		// 3. Lateral nicht OK: Querrichtung bevorzugen, Einfahrt gedrosselt
		ELSIF (PosLatOK = FALSE) THEN
			IF ePocketOrientation = ePocketX THEN
				FB_Positionsregler(targetPos := targetPos, actualPos := actualPos,
								KPX := 0.2 * KPX, KPY := KPY, KIX := 0.2 * KIX, KIY := KIY,
								vXCartesianToMotors     => targetSpeed_Robot.reX,
								vYCartesianToMotors     => targetSpeed_Robot.reY,
								vThetaCartesianToMotors => targetSpeed_Robot.reWinkel);
			ELSE
				FB_Positionsregler(targetPos := targetPos, actualPos := actualPos,
								KPX := KPX, KPY := 0.1 * KPY, KIX := KIX, KIY := 0.1 * KIY,
								vXCartesianToMotors     => targetSpeed_Robot.reX,
								vYCartesianToMotors     => targetSpeed_Robot.reY,
								vThetaCartesianToMotors => targetSpeed_Robot.reWinkel);
			END_IF
			GVL_Datatransfer23.inStatus := RobotStatus.laufend;
		
		// 4. Normalbetrieb
		ELSIF (Gripper.slider = TRUE) THEN
			
			IF ePocketOrientation = ePocketX THEN
				FB_Positionsregler(targetPos := targetPos, actualPos := actualPos,
								KPX := KPX, KPY := KPY, KIX := KIX, KIY := KIY,
								vXCartesianToMotors     => targetSpeed_Robot.reX,
								vYCartesianToMotors     => targetSpeed_Robot.reY,
								vThetaCartesianToMotors => targetSpeed_Robot.reWinkel);
			ELSE
				FB_Positionsregler(targetPos := targetPos, actualPos := actualPos,
								KPX := KPX, KPY := KPY, KIX := KIX, KIY := 2*KIY,
								vXCartesianToMotors     => targetSpeed_Robot.reX,
								vYCartesianToMotors     => targetSpeed_Robot.reY,
								vThetaCartesianToMotors => targetSpeed_Robot.reWinkel);
			END_IF			
			GVL_Datatransfer23.inStatus := RobotStatus.laufend;
		
		// 5. Ziel erreicht
		ELSE
			FB_Positionsregler(targetPos := targetPos, actualPos := actualPos,
								vXCartesianToMotors     => targetSpeed_Robot.reX,
								vYCartesianToMotors     => targetSpeed_Robot.reY,
								vThetaCartesianToMotors => targetSpeed_Robot.reWinkel);
								targetSpeed_Robot.reY := 0;
								targetSpeed_Robot.reX := 0;
								targetSpeed_Robot.reWinkel := 0;
			GVL_Datatransfer23.inStatus := RobotStatus.zielErreicht;
		END_IF
	
	END_CASE
	
//enableMotorControl := FALSE;
/////////////////////////////////////////////////////////////////////////////////////////////////////////
// Drehzahlregler
/////////////////////////////////////////////////////////////////////////////////////////////////////////
FB_Drehzahlregler(targetVelX			:= targetSpeed_Robot.reX,
					targetVelY 			:= targetSpeed_Robot.reY, 
					tragetVelTheta		:= targetSpeed_Robot.reWinkel,
					enable 				:= enableMotorControl,
					bumper 				:= bumper,
					MotorReset 			:= FALSE,
					actualVelMotor1 	:= -velWheel1, 
					actualVelMotor2 	:= -velWheel2, 
					actualVelMotor3 	:= -velWheel3,
					enableToMotor1 		=> enableToMotor1,
					enableToMotor2 		=> enableToMotor2,
					enableToMotor3 		=> enableToMotor3,
					velocityToMotor1	=> velocityToMotor1, 
					velocityToMotor2	=> velocityToMotor2,
					velocityToMotor3	=> velocityToMotor3);

ACTION ACT_Drehzahlerfassung:
//Einlesen der Istwerte
//Motorstrom von der Klemme auslesen und umrechnen
Motor1current := UINT_TO_INT(currentfromMotor1);	//Umwandlung des Unsinged Integers in ein Integerwert
Motor2current := UINT_TO_INT(currentfromMotor2);
Motor3current := UINT_TO_INT(currentfromMotor3);

//Berechnung der Radgeschwindigkeit mit berücksichtigung des Getriebes
velWheel1 := -(UINT_TO_INT(n1fromMotor) / maxKlemmeDrehzahlMessung*maxMotorRPM/60*ue*2*PI*rWheel);
velWheel2 := -(UINT_TO_INT(n2fromMotor) / maxKlemmeDrehzahlMessung*maxMotorRPM/60*ue*2*PI*rWheel);
velWheel3 := -(UINT_TO_INT(n3fromMotor) / maxKlemmeDrehzahlMessung*maxMotorRPM/60*ue*2*PI*rWheel);
END_ACTION

METHOD ATAN2 : LREAL
VAR_INPUT
    y : LREAL;
    x : LREAL;
END_VAR

VAR
    raw_angle : LREAL;
END_VAR

IF x = 0.0 THEN
    IF y > 0.0 THEN
        ATAN2 := 90.0;
    ELSIF y < 0.0 THEN
        ATAN2 := 270.0;
    ELSE
        ATAN2 := 0.0;
    END_IF;

ELSE
    raw_angle := ATAN(y / x) * (180.0 / PI);

    IF x > 0.0 THEN
        ATAN2 := raw_angle;
    ELSE
        ATAN2 := raw_angle + 180.0;
    END_IF;

    IF ATAN2 < 0.0 THEN
        ATAN2 := ATAN2 + 360.0;
    END_IF;
END_IF;
END_METHOD

METHOD Beobachter
VAR_INPUT
	wheelSpeed : WheelVelocity;
	cameraData : CameraConnectionUDP;
	RobotIndex : INT;
END_VAR
VAR_OUTPUT
	eastPos : sPosition := (reX := 0, reY := 0, reWinkel := 0);
END_VAR
VAR CONSTANT
	// === BEOBACHTER-PARAMETER => Großer Gain bedeutet hohes vertrauen in Kamera ===
	L_Gain					: REAL := 1.0;			// Luenberger Gain für X 		(0.0001-0.1)

	CYCLETIME 				: LREAL := 0.00033333;  // Cycletime des Motortasks
	CAMERA_DELAY			: REAL 	:= 0.1;
	BUFFWE_LENGTH			: INT 	:= 500;
	CAMERA_ERROR_THRESHOLD	: REAL 	:= 5.0;		// Fehlergrenze
	CAMERA_TIMEOUT			: LREAL := 30.0;		// Timeout in Sekunden
END_VAR

VAR_STAT
	bufferWheelSpeed	: ARRAY[0..BUFFWE_LENGTH] OF WheelVelocity;			// Speichern der letzten 300 Motorwerte (entspricht 100 ms -> Delay)
	prefCamPos			: sPosition;			// vorherige Kamera Position
	camPos				: sPosition;
	modelPos			: sPosition;
	CurrentTime			: LREAL;
	CameraTimestamp		: LREAL;
	actualError			: LREAL;				// Kamerafehler
	bufferIdx			: INT := 0;
	init				: BOOL;
END_VAR
VAR
	P_currentState 		: ARRAY[1..9] OF LREAL;	// Wär später für Kalmann	
	i					: INT;					// Iterrationsvariable
	averageWheelSpeed 	: WheelVelocity;
	x_estimated			: INT;
	angleError			: LREAL;
	idx					: INT;
	steps				: INT;
	startIdx			: INT;
	variableGain		: LREAL;
END_VAR
// Am anfang einmal die Kammeraposition direkt übertragen
IF init = TRUE THEN
	// Wenn ein guter Kamerawert gefunden wurde direkt einmal übertragen
	IF cameraData.robotPosition[RobotIndex].e < CAMERA_ERROR_THRESHOLD THEN
		camPos.reX 			:= cameraData.robotPosition[RobotIndex].x;
		camPos.reY 			:= cameraData.robotPosition[RobotIndex].y;
		camPos.reWinkel 	:= cameraData.robotPosition[RobotIndex].theta;
		actualError			:= cameraData.robotPosition[RobotIndex].e;
		prefCamPos 	:= camPos;
		modelPos	:= camPos;
		eastPos		:= camPos;
		
		init := FALSE;
	END_IF
ELSE
	/////////////////////////////////////////////////////////////////////////////////////////////////////////
	// Radwerte in FIFO abspeichern
	/////////////////////////////////////////////////////////////////////////////////////////////////////////
	bufferWheelSpeed[bufferIdx] := wheelSpeed;
	bufferIdx := (bufferIdx + 1) MOD BUFFWE_LENGTH;
	
	/////////////////////////////////////////////////////////////////////////////////////////////////////////
	// Modell Propagieren
	/////////////////////////////////////////////////////////////////////////////////////////////////////////
	propagate_state(
				X_Start 	:= modelPos,
				wheelSpeed 	:= wheelSpeed, 
				P_Start 	:= P_currentState,
				deltaT 		:= CYCLETIME,
				X_Predict 	=> modelPos,
				P_Predict 	=> P_currentState
			);
	CurrentTime := CurrentTime + CYCLETIME;	// Zeit weiter laufen lassen, wenn keine Kameradaten kommen
	
	/////////////////////////////////////////////////////////////////////////////////////////////////////////
	// Kameradaten verarbeiten
	/////////////////////////////////////////////////////////////////////////////////////////////////////////
	
	// Kammeraposition erst validieren
	IF cameraData.robotPosition[RobotIndex].e > CAMERA_ERROR_THRESHOLD OR
		// Prüfen ob neue Kameraposition
	   ((prefCamPos.reX 	 = cameraData.robotPosition[RobotIndex].x)	AND
		(prefCamPos.reY 	 = cameraData.robotPosition[RobotIndex].y) 	AND
		(prefCamPos.reWinkel = cameraData.robotPosition[RobotIndex].theta)) THEN
			
			// Falls keine neue Kameraposition erscheint, auch die Kamera vorwärtspropagieren
			propagate_state(
					X_Start 	:= camPos,
					wheelSpeed 	:= wheelSpeed, 
					P_Start 	:= P_currentState,
					deltaT 		:= CYCLETIME,
					X_Predict 	=> camPos,
					P_Predict 	=> P_currentState
				);
	ELSE
		// Falls Kameraposition gut nehmen
		camPos.reX 			:= cameraData.robotPosition[RobotIndex].x;
		camPos.reY 			:= cameraData.robotPosition[RobotIndex].y;
		camPos.reWinkel 	:= cameraData.robotPosition[RobotIndex].theta;
		actualError			:= cameraData.robotPosition[RobotIndex].e;
		CameraTimestamp 	:= (cameraData.HH * 60 + cameraData.MM) * 60 + cameraData.SS;
		CurrentTime			:= CameraTimestamp;
		
		// Abspeichern der actualposition als alte Kameraposition

		prefCamPos := camPos;
		
		// Alle Werte zurückrechnen
		steps := LREAL_TO_INT(CAMERA_DELAY / CYCLETIME);
		startIdx := bufferIdx - steps;
		IF startIdx < 0 THEN
			startIdx := startIdx + BUFFWE_LENGTH;
		END_IF
			
		FOR i := 0 TO steps - 1 DO
			idx := startIdx + i;
			IF idx >= BUFFWE_LENGTH THEN
				idx := idx - BUFFWE_LENGTH;
			END_IF
		

			propagate_state(
				X_Start 	:= camPos,
				wheelSpeed 	:= bufferWheelSpeed[idx], 
				P_Start 	:= P_currentState,
				deltaT 		:= CYCLETIME,
				X_Predict 	=> camPos,
				P_Predict 	=> P_currentState
			);
		END_FOR	
	END_IF	
	
	/////////////////////////////////////////////////////////////////////////////////////////////////////////
	// LUENBERGER-KORREKTUR: x_hat = x_model + L * (y - x_model)
	/////////////////////////////////////////////////////////////////////////////////////////////////////////
// 	variableGain := L_Gain * actualError/CAMERA_ERROR_THRESHOLD;
// 	IF variableGain > 1 OR variableGain < 0.0001 THEN
// 		variableGain := L_Gain;
// 	END_IF
// 	eastPos.reX 	 	:= modelPos.reX 		+ variableGain 	*	(camPos.reX 		- modelPos.reX);
// 	eastPos.reY 	 	:= modelPos.reY 		+ variableGain 	*	(camPos.reY 		- modelPos.reY);
// 	eastPos.reWinkel 	:= modelPos.reWinkel 	+ variableGain 	*	 NormalizeAngle(camPos.reWinkel - modelPos.reWinkel);

	eastPos.reX 	 	:= modelPos.reX 		+ L_Gain 	*	(camPos.reX 		- modelPos.reX);
	eastPos.reY 	 	:= modelPos.reY 		+ L_Gain 	*	(camPos.reY 		- modelPos.reY);
	eastPos.reWinkel 	:= modelPos.reWinkel 	+ L_Gain 	*	 NormalizeAngle(camPos.reWinkel - modelPos.reWinkel);
	modelPos := eastPos;
END_IF
END_METHOD

METHOD GetMinDistance : LREAL
VAR_INPUT
    velAngle    : LREAL;
    tolerance   : LREAL;
END_VAR
VAR
    i              : INT;
    sensorAngle    : LREAL;
    diff           : LREAL;
    minDistance    : LREAL := 1.0E+38;
END_VAR

FOR i := 1 TO 9 DO
    sensorAngle := (i - 1) * 40.0;

    diff := sensorAngle - velAngle;

    IF diff > 180.0 THEN
        diff := diff - 360.0;
    ELSIF diff < -180.0 THEN
        diff := diff + 360.0;
    END_IF;

    IF ABS(diff) <= tolerance THEN
        minDistance := MIN(minDistance, IrDistanceSensors.distance_mm[i]);
    END_IF;
END_FOR;

GetMinDistance := minDistance;
END_METHOD

METHOD NormalizeAngle
VAR_INPUT
	angle : LREAL;
END_VAR
VAR_OUTPUT
	NormalizeAngle :LREAL;
END_VAR
WHILE angle > PI DO
    angle := angle - (2.0 * PI);
END_WHILE

WHILE angle < -PI DO
    angle := angle + (2.0 * PI);
END_WHILE

NormalizeAngle := angle;
END_METHOD

METHOD propagate_state
VAR_INPUT
	X_Start 	: sPosition;
    wheelSpeed 	: WheelVelocity;   (* w1,w2,w3 *)
	P_Start 	: ARRAY[1..9] OF LREAL;
	deltaT 		: LREAL;
END_VAR

VAR_OUTPUT
    X_Predict : sPosition;
	P_Predict : ARRAY[1..9] OF LREAL;
END_VAR

VAR
    (* Body velocities *)
    bodyVelX : LREAL;
    bodyVelY : LREAL;
    yawRate  : LREAL;

    (* Weltkoordinaten Geschw. *)
    worldVelX : LREAL;
    worldVelY : LREAL;

    (* Jacobian Elemente *)
    jac13 : LREAL;
    jac23 : LREAL;

    (* Diskrete Übergangsterme *)
    a13 : LREAL;
    a23 : LREAL;

    (* Prozessrauschen *)// Muss noch gemessen werden => Abweichen der Räder
    qx : LREAL := 0.001;
    qy : LREAL := 0.001;
    qyaw : LREAL := 0.001;
END_VAR
(* ========================================================= *)
(*  EKF PREDICTION STEP – 3 Wheel Omni Robot                *)
(*  Zustandsvektor: x = [posX, posY, yaw]                   *)
(*  Modell: rein kinematisch                                 *)
(*  Diskretisierung: Vorwärts-Euler                          *)
(* ========================================================= *)

X_Start.reWinkel := -X_Start.reWinkel;

(* --- Wheel -> Body --- *)
bodyVelX := -(2.0/3.0) * (
			   -SIN(60  * PI/180) * wheelSpeed.wheel1
			   -SIN(180 * PI/180) * wheelSpeed.wheel2
			   -SIN(300 * PI/180) * wheelSpeed.wheel3
		   );

bodyVelY := -(2.0/3.0) * (
				COS(60  * PI/180) * wheelSpeed.wheel1
			  + COS(180 * PI/180) * wheelSpeed.wheel2
			  + COS(300 * PI/180) * wheelSpeed.wheel3
		   );

yawRate := -(wheelSpeed.wheel1 + wheelSpeed.wheel2 + wheelSpeed.wheel3) 
		   / (3.0 * GVL_RobotConstant.ROBOT_RADIUS * 1000);// Umrechnung in mm

(* --- Body -> World --- *)
worldVelX := bodyVelX * COS(X_Start.reWinkel)
		   - bodyVelY * SIN(X_Start.reWinkel);

worldVelY := bodyVelX * SIN(X_Start.reWinkel)
		   + bodyVelY * COS(X_Start.reWinkel);


(* --- Integration --- *)
X_Predict.reX 		:= X_Start.reX + deltaT * worldVelX;
X_Predict.reY 		:= X_Start.reY + deltaT * worldVelY;
X_Predict.reWinkel 	:= X_Start.reWinkel + deltaT * yawRate;


(* --- Winkel normalisieren --- *)

NormalizeAngle(angle := X_Predict.reWinkel, NormalizeAngle => X_Predict.reWinkel);

X_Predict.reWinkel := - X_Predict.reWinkel;


P_Predict := P_Start;
(*
(* ========================================================= *)
(* 4) Jacobi-Matrix F = ∂f/∂x                                *)
(*    Nur Ableitung nach yaw ist ≠ 0                         *)
(* ========================================================= *)

(* kontinuierliche Jacobi-Elemente *)

jac13 := -bodyVelX * SIN(X_Predict.reWinkel)
         -bodyVelY * COS(X_Predict.reWinkel);

jac23 :=  bodyVelX * COS(X_Predict.reWinkel)
         -bodyVelY * SIN(X_Predict.reWinkel);



(* ========================================================= *)
(* 5) Diskretisierung der Systemmatrix                       *)
(*    F_d = I + F*dt (Euler-Näherung)                        *)
(* ========================================================= *)

a13 := jac13 * deltaT;   (* entspricht F_d(1,3) *)
a23 := jac23 * deltaT;   (* entspricht F_d(2,3) *)



(* ========================================================= *)
(* 6) Kovarianz-Prediction                                   *)
(*    P = F_d * P * F_d^T + Q_d                              *)
(*                                                            *)
(*    P ist symmetrisch gespeichert:                          *)
(*    [ p11 p12 p13                                           *)
(*      p12 p22 p23                                           *)
(*      p13 p23 p33 ]                                         *)
(* ========================================================= *)

(* ---- Zwischenergebnis F_d * P * F_d^T ---- *)

P_Predict[1] := P_Start[1] + a13*(2.0*P_Start[3] + a13*P_Start[9]);
P_Predict[2] := P_Start[2] + a13*P_Start[6] + a23*P_Start[3] + a13*a23*P_Start[9];
P_Predict[3] := P_Start[3] + a13*P_Start[9];

P_Predict[5] := P_Start[5] + a23*(2.0*P_Start[6] + a23*P_Start[9]);
P_Predict[6] := P_Start[6] + a23*P_Start[9];

P_Predict[9] := P_Start[9];   (* yaw-Unsicherheit wächst nur durch Q *)



(* ========================================================= *)
(* 7) Prozessrauschen addieren                               *)
(*    Q_d = Q * dt                                           *)
(* ========================================================= *)

P_Predict[1] := P_Predict[1] + qx   * deltaT;
// P_Predict[2] := P_Predict[2];
// P_Predict[3] := P_Predict[3];

P_Predict[5] := P_Predict[5] + qy   * deltaT;
// P_Predict[6] := P_Predict[6];

P_Predict[9] := P_Predict[9] + qyaw * deltaT;
*)
END_METHOD

END_PROGRAM

// ---- POUs/HAWinoCore/001_MotorTask/FB_Drehzahlregler.TcPOU
FUNCTION_BLOCK FB_Drehzahlregler
VAR_INPUT
//Inputs: CartesianToMotors + Bumper
	targetVelX 	:	LREAL;			//Geschwindigkeitsvorgabe in X-Richtung im Robotersystem
	targetVelY 	:	LREAL;			//Geschwindigkeitsvorgabe in Y-Richtung im Robotersystem
	tragetVelTheta :	LREAL; 		//Geschwindigkeitsvorgabe in theta-Richtung im Robotersystem
	actualVelMotor1 : LREAL;			//Aktuelle Motordrehzahl Motor 1
	actualVelMotor2 : LREAL;			//Aktuelle Motordrehzahl Motor 2
	actualVelMotor3 : LREAL;			//Aktuelle Motordrehzahl Motor 3		
	enable 			 : BOOL;	//Freigabe des Reglers
	bumper	 		: BOOL;	
	MotorReset		: BOOL;		//Initialisieren des Reglers
END_VAR
VAR_OUTPUT
	//Outputs: Motor Values and Enable Signal
	enableToMotor1 :BOOL:=FALSE;		//Freigabe Motor 1 zur Klemme
	enableToMotor2 :BOOL:=FALSE;		//Freigabe Motor 2 zur Klemme
	enableToMotor3 :BOOL:=FALSE;		//Freigabe Motor 3 zur Klemme
		
	velocityToMotor1 :INT:=0;			//Geschwindigkeit zum Motor 1
	velocityToMotor2 :INT:=0;			//Geschwindigkeit zum Motor 2
	velocityToMotor3 :INT:=0;			//Geschwindigkeit zum Motor 3
END_VAR
VAR
	//Umgerechnete Werte
	vX:		LREAL:=0;	//Inverse Sollgeschwindigkeit in X-Richtung		
	vY:		LREAL:=0;	//Inverse Sollgeschwindigkeit in Y-Richtung	
	vTheta:	LREAL:=0;	//Inverse Sollgeschwindigkeit in Theta-Richtung	

	//Fahrrichtung Motor
	targetVelocityMotor1: LREAL;	//Sollgeschwindigkeit für Motor 1
	targetVelocityMotor2: LREAL;	//Sollgeschwindigkeit für Motor 2
	targetVelocityMotor3: LREAL;	//Sollgeschwindigkeit für Motor 3
	
	//Skalierung auf MaxGeschwindigkeit Skalierung hängt mit CoE Register 8020:07 8020:08 zusammen !!!
	velocityMax:LREAL:=942.4777961;// Nenndrehzahl U/min CoE Register 8020:07 8020:08 fesgelegt Faktor 16 Wegen Getriebe 1:16
	velocityMotorsTf:LREAL:=0;		//Hilfsvariable zur Begrenzung der Radgeschwindigkeiten
	
	// Skalierung auf Ansteuersignale LREAL=>WORD   Skalierung hängt mit CoE Register 8020:07 8020:08 zusammen !!!
	skalPos:LREAL:=34.7668668;//  MaxValue/MaxVelocity   [1/ mm/s]   32767/(942mm/s)   MaxVelocity=D*PI*n/(16*60) //16:1 Getriebeübersetzung  
	skalNeg:LREAL:=34.76792783;//  MaxVelau/MaxVelocity   [1/ mm/s]   32768/(942mm/s)   MaxVelocity=(80mm*PI*3600 U/min)/(16*60sec/min)
	
	//Reglerwerte
	errorM1: LREAL;	//Regeldifferenz Motor 1
	errorM2: LREAL;	//Regeldifferenz Motor 2
	errorM3: LREAL;	//Regeldifferenz Motor 3
	
	IntegralM1 : LREAL :=0;	//Integrator Motor 1
	IntegralM2 : LREAL :=0;	//Integrator Motor 2
	IntegralM3 : LREAL :=0;	//Integrator Motor 3
	
	LastIntegralM1 : LREAL := 0;
	LastIntegralM2 : LREAL := 0;
	LastIntegralM3 : LREAL := 0;
	
	velocityM1Controled: LREAL;	//Geregelte geschwindigkeitsansteuerung Motor 1
	velocityM2Controled: LREAL;	//Geregelte geschwindigkeitsansteuerung Motor 2
	velocityM3Controled: LREAL;	//Geregelte geschwindigkeitsansteuerung Motor 3
	
	KP : REAL :=1; 	//P Anteil des Reglers
	KI : REAL :=214;		//I Anteil des Reglers
	
	//Zustandsautomat des Reglers
	state: ReglerState :=	ReglerState.init;
	nCycleTime: UDINT;
	fbGetCurTaskIdx: GETCURTASKINDEX;
	index: INT;
	diffConst: LREAL :=1; //Zykluszeit für die Integratoren. Wird dynamisch bestimmt

	testtargetVelXRobo		: LREAL;
	testtargetVelYRobo		: LREAL;
	testtragetVelThetaRobo	: LREAL;
END_VAR

//Aufrufen des Zustandsautomats des Reglers
ACT_Zustandsautomat();

//Invertieren der Sollgeschwindigkeiten
vX 		:= -targetVelX;
vY 		:= -targetVelY;
vTheta	:= -tragetVelTheta;
// vx := -100;
// vY := 00;
// vTheta:= 1;

//Umrechnung der Kartesischen Geschwindigkeit auf die einzelnen Motoren
// targetVelocityMotor1 := ((-vX * COS(30.0*PI/180))	+ (vY * COS(60.0*PI/180))	+ (vTheta * 135.0));
// targetVelocityMotor2 := (0.0							+ (-vY)						+ (vTheta * 135.0));
// targetVelocityMotor3 := ((vX * COS(30.0*PI/180))		+ (vY * COS(60.0*PI/180))	+ (vTheta * 135.0));

targetVelocityMotor1 := -SIN(60  * PI/180) * vX + COS(60  * PI/180) * vY + GVL_RobotConstant.ROBOT_RADIUS * 1000 * vTheta; // Robot Radius in mm umrechnen
targetVelocityMotor2 := -SIN(180 * PI/180) * vX + COS(180 * PI/180) * vY + GVL_RobotConstant.ROBOT_RADIUS * 1000 * vTheta;
targetVelocityMotor3 := -SIN(300 * PI/180) * vX + COS(300 * PI/180) * vY + GVL_RobotConstant.ROBOT_RADIUS * 1000 * vTheta;

//Begrenzung der Sollwerte und anpassung aller Sollvorgaben an den Motor mit der Maximalen geschwindigkeit
ACT_Sollwertbegrenzung();

//Regleung der einzelnen Motoren
//Differenzbildung der Drehzahlen
errorM1 := targetVelocityMotor1 - actualVelMotor1;
errorM2 := targetVelocityMotor2 - actualVelMotor2;
errorM3 := targetVelocityMotor3 - actualVelMotor3;

//Integratoren der Motoren
IntegralM1 := IntegralM1 + (errorM1 * diffConst);
IntegralM2 := IntegralM2 + (errorM2 * diffConst);
IntegralM3 := IntegralM3 + (errorM3 * diffConst);

//Zusammenführung der P und I Anteile der Motoren
velocityM1Controled := (errorM1 *KP) + (KI *IntegralM1);
velocityM2Controled := (errorM2 *KP) + (KI *IntegralM2);
velocityM3Controled := (errorM3 *KP) + (KI *IntegralM3);

//Löschen des Integrators, wenn die Sollposition erreicht ist, da sonst eine Restansteuerung bleibt
ACT_ResetIntegrators();
//Begrenzung der Ansteuerung auf den maximalen Wert
ACT_Ansteuerungsbegrenzung();

ACTION ACT_Ansteuerungsbegrenzung:
//Begrenzung der Ansteuerung
// Wenn die berechnete Geschwindigkeit von Motor 1 (velocityM1Controled) größer als die maximal zulässige Geschwindigkeit (velocityMax) ist,
// wird die Geschwindigkeit auf den maximalen Wert begrenzt und der Integralwert (IntegralM1) auf den letzten gespeicherten Wert zurückgesetzt.
IF ( velocityM1Controled > velocityMax) THEN
	velocityM1Controled := velocityMax;
	IntegralM1 := LastIntegralM1;
// Wenn die berechnete Geschwindigkeit kleiner als die negative maximale Geschwindigkeit ist,
// wird sie auf den minimalen Wert (-velocityMax) begrenzt und der Integralwert eingefroren.
ELSIF(velocityM1Controled < -velocityMax) THEN
	velocityM1Controled := -velocityMax;
	IntegralM1 := LastIntegralM1;

ELSE
// Wenn die berechnete Geschwindigkeit innerhalb des zulässigen Bereichs liegt,
// wird der aktuelle Integralwert gespeichert.
	LastIntegralM1 := IntegralM1;		
END_IF

// Begrenzung der Ansteuerung für Motor 2
//Selbe Logik wie bei Motor 1
IF ( velocityM2Controled > velocityMax) THEN
	velocityM2Controled := velocityMax;
	IntegralM2 := LastIntegralM2;
ELSIF(velocityM2Controled < -velocityMax) THEN
	velocityM2Controled := -velocityMax;
	IntegralM2 := LastIntegralM2;
ELSE
	LastIntegralM2 := IntegralM2;
END_IF

// Begrenzung der Ansteuerung für Motor 3
//Selbe Logik wie bei Motor 1
IF ( velocityM3Controled > velocityMax) THEN
	velocityM3Controled := velocityMax;
	IntegralM3 := LastIntegralM3;
ELSIF(velocityM3Controled < -velocityMax) THEN
	velocityM3Controled := -velocityMax;
	IntegralM3 := LastIntegralM3;
ELSE
	LastIntegralM3 := IntegralM3;
END_IF
END_ACTION

ACTION ACT_ResetIntegrators:

//Löschen des Integrators beim Stillstand, da die Motoren sonst brummen
IF ABS(errorM1) < 0.02 AND ABS(targetVelocityMotor1) < 0.02 THEN
		IntegralM1 :=0;
END_IF
IF ABS(errorM2) < 0.02 AND ABS(targetVelocityMotor2) < 0.02 THEN
		IntegralM2 :=0;
END_IF
IF ABS(errorM3) < 0.02 AND ABS(targetVelocityMotor3) < 0.02 THEN
		IntegralM3 :=0;
END_IF
END_ACTION

ACTION ACT_Sollwertbegrenzung:


//Begrenzung der Maximalen Soll-Drehzahl
//Überprüfung der Sollwerte für Motor 1
IF (ABS(targetVelocityMotor1) > velocityMax)THEN	//Ueberpruefen, ob die Absolute Sollgeschwindigkeit über der Maximalen ist
	velocityMotorsTf:= targetVelocityMotor1; 		//Speichern der erwünschten Geschwindigkeit
    targetVelocityMotor1:= velocityMotorsTf/ABS(velocityMotorsTf)*velocityMax;		//Begrenzung auf die Maximale Geschwindigkeit
    targetVelocityMotor2:= velocityMotorsTf/ABS(velocityMotorsTf)*velocityMax/velocityMotorsTf * targetVelocityMotor2 ;		//Verhältnissmäßige anpassung der Geschwindigkeit
    targetVelocityMotor3:= velocityMotorsTf/ABS(velocityMotorsTf)*velocityMax/velocityMotorsTf * targetVelocityMotor3 ;		//Verhältnissmäßige anpassung der Geschwindigkeit
END_IF

//Überprüfung der Sollwerte für Motor 2
IF (ABS(targetVelocityMotor2) > velocityMax)THEN	//Ueberpruefen, ob die Absolute Sollgeschwindigkeit über der Maximalen ist
    velocityMotorsTf:= targetVelocityMotor2;		//Speichern der erwünschten Geschwindigkeit
     targetVelocityMotor1:= velocityMotorsTf/ABS(velocityMotorsTf)*velocityMax/velocityMotorsTf * targetVelocityMotor1;		//Verhältnissmäßige anpassung der Geschwindigkeit
    targetVelocityMotor2:= velocityMotorsTf/ABS(velocityMotorsTf)*velocityMax;		//Begrenzung auf die Maximale Geschwindigkeit
    targetVelocityMotor3:= velocityMotorsTf/ABS(velocityMotorsTf)*velocityMax/velocityMotorsTf * targetVelocityMotor3;		//Verhältnissmäßige anpassung der Geschwindigkeit
END_IF

//Überprüfung der Sollwerte für Motor 3	
IF (ABS(targetVelocityMotor3) > velocityMax) THEN	//Ueberpruefen, ob die Absolute Sollgeschwindigkeit über der Maximalen ist
    velocityMotorsTf:= targetVelocityMotor3;		//Speichern der erwünschten Geschwindigkeit
    targetVelocityMotor1:= velocityMotorsTf/ABS(velocityMotorsTf)*velocityMax/velocityMotorsTf * targetVelocityMotor1;		//Verhältnissmäßige anpassung der Geschwindigkeit
    targetVelocityMotor2:= velocityMotorsTf/ABS(velocityMotorsTf)*velocityMax/velocityMotorsTf * targetVelocityMotor2 ;		//Verhältnissmäßige anpassung der Geschwindigkeit
    targetVelocityMotor3:= velocityMotorsTf/ABS(velocityMotorsTf)*velocityMax;		//Begrenzung auf die Maximale Geschwindigkeit
END_IF
END_ACTION

ACTION ACT_Zustandsautomat:

//Rücksetzen des Zustandsautomaten
IF MotorReset THEN
	state := ReglerState.init;
END_IF

//MOTORANSTEUERUNG Zustandsautomat
CASE state OF
	ReglerState.init:	
		//GetCycletime Motortask	
		fbGetCurTaskIdx();
		nCycleTime := _TaskInfo[fbGetCurTaskIdx.index].CycleTime; //multiplier of 100ns
		diffConst := UDINT_TO_LREAL(nCycleTime) * 0.0000001; //
		
		//Ansteuerung der Motoren abschalten
		velocityToMotor1:=0;
		velocityToMotor2:=0;
		velocityToMotor3:=0;
		//Freigabe der Motoren entziehen
		enableToMotor1:=0;
		enableToMotor2:=0;
		enableToMotor3:=0;
		//Integratoren zurücksetzen
		IntegralM1 :=0;
		IntegralM2 :=0;
		IntegralM3 :=0;
		//Wechsel in den Idle zustand
		state:=ReglerState.idle;
		
	ReglerState.idle:
		//Wenn die Fahrtfreigabe erteilt ist, wechselt der Regler in working
		IF enable THEN
			state := ReglerState.working;
		END_IF	
		//Wenn der Bumper ausgelöst hat, Wechselt der Motor in Stop	
		IF bumper THEN
			state:=ReglerState.stop;
		END_IF
		//Abschalten der Motoransteuerung
		velocityToMotor1:=0;
		velocityToMotor2:=0;
		velocityToMotor3:=0;
		//Entzug der Motorenfreigabe
		enableToMotor1:=0;
		enableToMotor2:=0;
		enableToMotor3:=0;
		//Zurücksetzen der Integratoren
		IntegralM1 :=0;
		IntegralM2 :=0;
		IntegralM3 :=0;
	
	ReglerState.working:
		//Ansteuerung der Ausgänge mit Skallierungsfaktor auf INT-Maximalwerte Werte.
		IF velocityM1Controled>=0 THEN
			velocityToMotor1:=LREAL_TO_INT(velocityM1Controled*skalPos);
		ELSE	//Ansteuerung mit Negativem Skallierungsfaktor für negativen Geschwindigkeiten
			velocityToMotor1:=LREAL_TO_INT(velocityM1Controled*skalNeg);
		END_IF
		IF velocityM2Controled>=0 THEN
			velocityToMotor2:=LREAL_TO_INT(velocityM2Controled*skalPos);
		ELSE	//Ansteuerung mit Negativem Skallierungsfaktor für negativen Geschwindigkeiten
			velocityToMotor2:=LREAL_TO_INT(velocityM2Controled*skalNeg);
		END_IF
		
		IF velocityM3Controled>=0 THEN
			velocityToMotor3:=LREAL_TO_INT(velocityM3Controled*skalPos);
		ELSE	//Ansteuerung mit Negativem Skallierungsfaktor für negativen Geschwindigkeiten
			velocityToMotor3:=LREAL_TO_INT(velocityM3Controled*skalNeg); 
		END_IF
		//Erteilen der Motorfreigaben
		enableToMotor1:=1;
		enableToMotor2:=1;
		enableToMotor3:=1;
		
		//Wechseln in den Idle Zustand, wenn die Freigabe entzogen wird.
		IF enable = FALSE THEN
			state:=ReglerState.idle;
		END_IF
		//Sofortiges umschalten in den Stop Zustand, wenn der Bumper ausgelöst hat
		IF bumper THEN
			state:=ReglerState.stop;
		END_IF
						
	ReglerState.stop:
		//Ansteuerung der Ausgänge abschalten
		velocityToMotor1:=0;
		velocityToMotor2:=0;
		velocityToMotor3:=0;
		//Motorfreigaben entzeihen
		enableToMotor1:=0;
		enableToMotor2:=0;
		enableToMotor3:=0;
		//Zurücksetzen der Integratoren
		IntegralM1 :=0;
		IntegralM2 :=0;
		IntegralM3 :=0;
		//Zustandswechsel in den Idle zustand, wenn der Bumper ordnungsgemäß zurückgesetzt wird.
		IF NOT bumper AND enable THEN
			state := ReglerState.idle;
		END_IF
	ELSE
		//Bei einem Unbestimmten zustand wird der Regler Inittialisiert
		state:= ReglerState.init;
END_CASE
END_ACTION

END_FUNCTION_BLOCK

// ---- POUs/HAWinoCore/001_MotorTask/FB_Positionsregler.TcPOU
FUNCTION_BLOCK FB_Positionsregler
VAR_INPUT
	targetPos		: sPosition;
	actualPos		: sPosition;
	KPX				: LREAL 	:= 0.0;
	KPY				: LREAL 	:= 0.0;
	KIX				: LREAL 	:= 0.0;
	KIY				: LREAL 	:= 0.0;
	
END_VAR
VAR_OUTPUT
	vXCartesianToMotors		: LREAL :=0;
	vYCartesianToMotors		: LREAL :=0;
	vThetaCartesianToMotors	: LREAL :=0;
END_VAR
VAR
	error		: sPosition;	// Positionsfehler
	deltaError	: sPosition;	// Fehlersteigung
	integralError : sPosition;
	diffConst: LREAL :=0.001;

	// Geschwindigkeit in Weltkoordinaten 
	W_X_targetSpeed		: LREAL; 
	W_Y_targetSpeed		: LREAL; 
	W_Theta_targetSpeed : LREAL;
	
	// Geschwindigkeit in Roboterkoordinaten
	R_X_targetSpeed		: LREAL;
	R_Y_targetSpeed		: LREAL;
	R_Theta_targetSpeed	: LREAL;
	
	// Reglerparameter
	//KPX		: LREAL 	:= 0.8;
	//KPY		: LREAL		:= 0.8;
	KPTheta	: LREAL 	:= 1.5;
	//KIX 	: LREAL 	:= 0.025;
	KITheta : LREAL 	:= 0.1;
	
	speedThreshold	: LREAL := 0.01; //Annäherung nur aktiv bei Abweichung > threshold
	AccelerationRate: LREAL := 5; 	//Höhere Werte = höhere Beschleunigung
	
	// Fuzzy Calkulation
	MembershipE : ARRAY[1..5] OF LREAL;
	MembershipDE : ARRAY[1..5] OF LREAL;
	i: INT;
	j: INT;
	ruleIdx: INT;
	weight: LREAL;
	numerator : LREAL := 0.0;
	denominator : LREAL := 0.0;
	initDone: BOOL := FALSE;
	
	RuleTable : ARRAY[1..5, 1..5] OF INT;
	OutputValue : ARRAY[1..5] OF REAL := [
        0.0,   // ZS
        0.25,  // PS
        0.5,   // PM
        0.75,  // PL
        1.0    // HL
    ];
	oldErrorTheta: LREAL;
END_VAR

// Wollte ich eigentlich oben machen, aber wollte er iwie nicht. Auf dauer noch ändern
IF NOT initDone THEN
    // RuleTable initialisieren (Zeile-für-Zeile), vermeidet statische Literal-Initialisierung
    RuleTable[1,1] := 5; RuleTable[1,2] := 5; RuleTable[1,3] := 4; RuleTable[1,4] := 4; RuleTable[1,5] := 3;
    RuleTable[2,1] := 4; RuleTable[2,2] := 4; RuleTable[2,3] := 4; RuleTable[2,4] := 3; RuleTable[2,5] := 2;
    RuleTable[3,1] := 4; RuleTable[3,2] := 4; RuleTable[3,3] := 3; RuleTable[3,4] := 2; RuleTable[3,5] := 4;
    RuleTable[4,1] := 4; RuleTable[4,2] := 3; RuleTable[4,3] := 2; RuleTable[4,4] := 2; RuleTable[4,5] := 1;
    RuleTable[5,1] := 3; RuleTable[5,2] := 2; RuleTable[5,3] := 2; RuleTable[5,4] := 1; RuleTable[5,5] := 1;

    OutputValue[1] := 0.0;
    OutputValue[2] := 0.25;
    OutputValue[3] := 0.5;
    OutputValue[4] := 0.75;
    OutputValue[5] := 1.0;
	
	integralError.reX := 0;
	integralError.reY := 0;
	integralError.reWinkel := 0;

	
    initDone := TRUE;
END_IF

// --------------------------------------------------
// Winkelfehlerberechnung (Theta)
// --------------------------------------------------

// Winkelabweichung zwischen Soll und Ist berechnen
error.reWinkel := targetPos.reWinkel - actualPos.reWinkel;

// Normierung der Winkelabweichung auf den Bereich [-PI, PI]
// → stellt sicher, dass immer der kürzeste Drehweg verwendet wird
IF error.reWinkel > PI THEN
    error.reWinkel := error.reWinkel - 2.0 * PI;
ELSIF error.reWinkel < -PI THEN
    error.reWinkel := error.reWinkel + 2.0 * PI;
END_IF;

// Alten Fehlerwert für die Ableitung speichern
oldErrorTheta := error.reWinkel;

// Aktuellen Winkelfehler setzen
// Vorzeichen ggf. an Drehrichtungskonvention anpassen
error.reWinkel := -error.reWinkel;

// Änderung des Fehlers (D-Anteil)
deltaError.reWinkel := error.reWinkel - oldErrorTheta;


// --------------------------------------------------
// Positionsfehlerberechnung (X, Y)
// --------------------------------------------------

// Fehleränderung berechnen (Differenz zum vorherigen Fehler)
deltaError.reX := error.reX - (targetPos.reX - actualPos.reX);
deltaError.reY := error.reY - (targetPos.reY - actualPos.reY);

// Aktuellen Positionsfehler berechnen
error.reX := targetPos.reX - actualPos.reX;
error.reY := targetPos.reY - actualPos.reY;

IF KIX = 0.0 THEN
integralError.reX := 0.0;
ELSE
integralError.reX := integralError.reX + (error.reX * diffConst);
END_IF

//integralError.reY := integralError.reY + (error.reY * diffConst);
//integralError.reWinkel := integralError.reWinkel + (error.reWinkel * diffConst);

// --------------------------------------------------
// Positionsregelung
// --------------------------------------------------

// ACT_GetFuzzyParam();

// Berechnung der Stellgröße
W_X_targetSpeed 	:= (error.reX 		* KPX) + (KIX * integralError.reX);
W_Y_targetSpeed 	:= (error.reY 		* KPY);
W_Theta_targetSpeed := (error.reWinkel 	* KPTheta) + (KITheta * integralError.reWinkel);

// Umrechnung von Welt in Motorcoordinaten
R_X_targetSpeed 	:= W_X_targetSpeed * COS(actualPos.reWinkel) - W_Y_targetSpeed * SIN(actualPos.reWinkel);
R_Y_targetSpeed 	:= W_Y_targetSpeed * COS(actualPos.reWinkel) + W_X_targetSpeed * SIN(actualPos.reWinkel);
R_Theta_targetSpeed := W_Theta_targetSpeed;

ACT_LimitACC();

ACTION ACT_GetFuzzyParam:
// Berechnen des Kx Reglers
METH_InputMembership(e := error.reX, outArr := MembershipE);
METH_InputMembership(e := deltaError.reX, outArr := MembershipDE);

// Defuzzyfication
FOR i := 1 TO 5 DO
    FOR j := 1 TO 5 DO
        weight := MembershipE[i] * MembershipDE[j];
        ruleIdx := RuleTable[i,j];

        numerator := numerator + weight * OutputValue[ruleIdx];
        denominator := denominator + weight;
    END_FOR
END_FOR

IF denominator > 0 THEN
    KPX := numerator / denominator;
ELSE
    KPX := 0.0; // fallback
END_IF

// Berechnen des Ky Reglers
METH_InputMembership(e := error.reY, 		outArr := MembershipE);
METH_InputMembership(e := deltaError.reY, 	outArr := MembershipDE);

// Defuzzyfication
FOR i := 1 TO 5 DO
    FOR j := 1 TO 5 DO
        weight := MembershipE[i] * MembershipDE[j];
        ruleIdx := RuleTable[i,j];

        numerator := numerator + weight * OutputValue[ruleIdx];
        denominator := denominator + weight;
    END_FOR
END_FOR

IF denominator > 0 THEN
    KPY := numerator / denominator;
ELSE
    KPY := 0.0; // fallback
END_IF
END_ACTION

ACTION ACT_LimitACC:
//Smoothes Annähern an den Sollwert, anpassbar über integrationRate
// x Werte 
IF ABS(vXCartesianToMotors - R_X_targetSpeed) > speedThreshold THEN   
    IF vXCartesianToMotors < R_X_targetSpeed THEN
        vXCartesianToMotors := vXCartesianToMotors + AccelerationRate * 0.01;  //Beschleunigung vorwärts
    ELSE
        vXCartesianToMotors := vXCartesianToMotors - AccelerationRate * 0.01;  //Beschleunigung rückwärts
    END_IF
END_IF
// y Werte 
IF ABS(vYCartesianToMotors - R_Y_targetSpeed) > speedThreshold THEN   
    IF vYCartesianToMotors < R_Y_targetSpeed THEN
        vYCartesianToMotors := vYCartesianToMotors + AccelerationRate * 0.01;  //Beschleunigung vorwärts
    ELSE
        vYCartesianToMotors := vYCartesianToMotors - AccelerationRate * 0.01;  //Beschleunigung rückwärts
    END_IF
END_IF
// Theta Werte 
IF ABS(vThetaCartesianToMotors - R_Theta_targetSpeed) > speedThreshold THEN   
    IF vThetaCartesianToMotors < R_Theta_targetSpeed THEN
        vThetaCartesianToMotors := vThetaCartesianToMotors + AccelerationRate * 0.01;  //Beschleunigung vorwärts
    ELSE
       vThetaCartesianToMotors := vThetaCartesianToMotors - AccelerationRate * 0.01;  //Beschleunigung rückwärts
    END_IF
END_IF
END_ACTION

METHOD METH_InputMembership
VAR_INPUT
	e	: LREAL;
END_VAR
VAR_IN_OUT
	outArr : ARRAY[1..5] OF LREAL;
END_VAR
// einfache dreieckige Memberships als Beispiel (anpassen an deine MF)
outArr[1] := MAX(0.0, ( -e - 0.5) / 0.5);      // NL (links)
outArr[2] := MAX(0.0, 1.0 - ABS(e + 0.5) / 0.75); // NS
outArr[3] := MAX(0.0, 1.0 - ABS(e) / 1.0);       // ZE
outArr[4] := MAX(0.0, 1.0 - ABS(e - 0.5) / 0.75); // PS
outArr[5] := MAX(0.0, (e - 0.5) / 0.5);        // PL
END_METHOD

END_FUNCTION_BLOCK

// ---- POUs/HAWinoCore/04_SystemManagment/PowerManager.TcPOU
PROGRAM PowerManager
VAR_INPUT
	RobotData : RobotInternalData;
END_VAR
VAR
	shutdownButton			AT%I*  : BOOL := FALSE;			//Button zum Ausschalten
	shutdownTrigger 		AT%Q*  : BOOL := FALSE;			//Zeitablauf, bis Robi ausschaltet
	batteryVoltageRaw  		AT%I*  : INT;					//unverabreitete gemessene Spannung
	scaleVoltage:	REAL := LREAL_TO_REAL(20/EXPT(2,16));	//Skalierungsfaktor, um auf verarbeitete Spannung zu kommen. 
	batteryVoltage_V		AT%Q*  : REAL;					//verarbeitete Spannung
	supplyCurrentRaw		AT%I* : INT;					//unverabreitete gemessener Strom
	supplyCurrent_A			AT%Q* : REAL; 					//verarbeiteter Strom

	shutdown: NT_Shutdown;									//Befehl zum Herunterfahren

	stMqtt_HAWino_IN		AT%Q*	: ST_PwrMgmt_HAWino_In;	//Link MQTT-DatenStruct

	// Variablen für EKF
	debug :BOOl :=TRUE;
	EKF_init						: BOOL := TRUE; // für ersten EKF Zustand
	(* Puffer um nur 1 mal die Sekunde rechnen zu müssen*)
	writeIndex						: INT := 0;
	I_buffer        				: ARRAY [0..199] OF REAL;	//Puffer für die letzten 200 I-Werte, muss angepasst werden auf die Sampletime
	V_buffer						: ARRAY [0..199] OF REAL;	//Puffer für die letzten 200 V-Werte, muss angepasst werden auf die Sampletime
	buffer_counter					: INT := 0;			// Counter für den Buffer falls Werte durch Verdrängung nicht geschreiben werden
	I_sum							: REAL := 0;			// Summe der Buffers für mean Berechnung				
	V_sum 							: REAL := 0;			// Summe der Buffers für mean Berechnung
	I_mean							: REAL := 0;			// mean Wert		
	V_mean							: REAL := 0;			// mean Wert
	i								: INT;					// Laufvariable für Schleifen
	
	(*LUT*)
	SOC_Table : ARRAY[1..201] OF REAL := [0,0.005,0.01,0.015,0.02,0.025,0.03,0.035,0.04,0.045,0.05,0.055,0.06,0.065,0.07,0.075,0.08,0.085,0.09,0.095,0.1,0.105,0.11,0.115,0.12,0.125,0.13,0.135,0.14,0.145,0.15,0.155,0.16,0.165,0.17,0.175,0.18,0.185,0.19,0.195,0.2,0.205,0.21,0.215,0.22,0.225,0.23,0.235,0.24,0.245,0.25,0.255,0.26,0.265,0.27,0.275,0.28,0.285,0.29,0.295,0.3,0.305,0.31,0.315,0.32,0.325,0.33,0.335,0.34,0.345,0.35,0.355,0.36,0.365,0.37,0.375,0.38,0.385,0.39,0.395,0.4,0.405,0.41,0.415,0.42,0.425,0.43,0.435,0.44,0.445,0.45,0.455,0.46,0.465,0.47,0.475,0.48,0.485,0.49,0.495,0.5,0.505,0.51,0.515,0.52,0.525,0.53,0.535,0.54,0.545,0.55,0.555,0.56,0.565,0.57,0.575,0.58,0.585,0.59,0.595,0.6,0.605,0.61,0.615,0.62,0.625,0.63,0.635,0.64,0.645,0.65,0.655,0.66,0.665,0.67,0.675,0.68,0.685,0.69,0.695,0.7,0.705,0.71,0.715,0.72,0.725,0.73,0.735,0.74,0.745,0.75,0.755,0.76,0.765,0.77,0.775,0.78,0.785,0.79,0.795,0.8,0.805,0.81,0.815,0.82,0.825,0.83,0.835,0.84,0.845,0.85,0.855,0.86,0.865,0.87,0.875,0.88,0.885,0.89,0.895,0.9,0.905,0.91,0.915,0.92,0.925,0.93,0.935,0.94,0.945,0.95,0.955,0.96,0.965,0.97,0.975,0.98,0.985,0.99,0.995,1];	
	OCV_Table : ARRAY[1..201] OF REAL := [9.65696,10.01568,10.37441,10.73313,11.09186,11.45058,11.80931,12.16804,12.52676,12.88347,13.15018,13.33744,13.47367,13.58107,13.66917,13.74054,13.79451,13.83336,13.86090,13.88392,13.90258,13.92009,13.93595,13.95171,13.96639,13.98137,13.99666,14.01189,14.02784,14.04310,14.05916,14.07404,14.09014,14.10651,14.12697,14.14870,14.17227,14.19292,14.21337,14.23219,14.25112,14.27003,14.28847,14.30634,14.32343,14.33906,14.35275,14.36473,14.37573,14.38692,14.39651,14.40639,14.41586,14.42488,14.43347,14.44160,14.44941,14.45687,14.46397,14.47031,14.47772,14.48429,14.49075,14.49709,14.50339,14.50955,14.51567,14.52193,14.52803,14.53355,14.53994,14.54523,14.55164,14.55699,14.56331,14.56836,14.57502,14.58032,14.58658,14.59161,14.59841,14.60361,14.61012,14.61503,14.62174,14.62710,14.63358,14.63897,14.64537,14.65146,14.65749,14.66364,14.66981,14.67611,14.68243,14.68885,14.69529,14.70195,14.70869,14.71604,14.72228,14.72929,14.73647,14.74380,14.75133,14.75903,14.76699,14.77517,14.78363,14.79204,14.80156,14.81106,14.82105,14.83162,14.84286,14.85485,14.86769,14.88158,14.89608,14.91097,14.92572,14.94016,14.95417,14.96765,14.98187,14.99617,15.01116,15.02629,15.04195,15.05725,15.07354,15.08894,15.10475,15.12022,15.13591,15.15113,15.16751,15.18265,15.19897,15.21487,15.23111,15.24744,15.26394,15.28064,15.29752,15.31459,15.33183,15.34929,15.36708,15.38570,15.40277,15.42091,15.43924,15.45767,15.47633,15.49512,15.51398,15.53298,15.55202,15.57071,15.59069,15.61009,15.62960,15.64923,15.66889,15.68864,15.70848,15.72865,15.74808,15.76854,15.78813,15.80895,15.82880,15.84926,15.86945,15.89020,15.91045,15.93127,15.95181,15.97293,15.99372,16.01512,16.03615,16.05766,16.07912,16.10064,16.12199,16.14414,16.16646,16.18855,16.21118,16.23379,16.25666,16.27972,16.30307,16.32667,16.35062,16.37489,16.40038,16.42706,16.45582];
	i_LUT      : INT;    // Laufvariable 
    diff       : REAL;    //Abstand zwischen aktuellem SOC und Tabellenwert 
    diff_min   : REAL;    //kleinster bisher gefundener Abstand 
    idx_min    : INT;     //Index des nächsten Wertes 
    OCV        : REAL;    //Ausgewählter OCV-Wert
    dVdSOC     : REAL;    //Spannungsänderung pro SOC-Schritt 
	
	(* EKF Zustände *)
    x_SOC    : REAL := 0.5;           //  SOC
	param_SOC : REAL := 0;			  // SOC zur parameter Parameter 	
    x_Vrc    : REAL := 0.0;           // RC-Kondensatorspannung (V)

	(* Kovarianzmatrix-P *)
    P11 : REAL := 1;     // Var(SOC)
    P12 : REAL := 0.0;
    P21 : REAL := 0.0;
    P22 : REAL := 1;     // Var(Vrc)

	(* Batterieparameter *)
    R0       : REAL := 0.086; 		// Init Wert (bei 60% SOC)
    R1       : REAL := 0.0174; 		// Init Wert (bei 60% SOC)
    C1       : REAL := 763; 		// Init Wert (bei 60% SOC)
    Qbatt    : REAL := 63000.0;      // 17.5Ah → 63000 As
    eta      : REAL := 1.0;
    dt_ekf   : REAL := 1.0;          // EKF einmal die sekunde

	(* Rauschvarianzen *)
    Qz       : REAL := (2e-5)*(2e-5);   // SoC Prozessrauschen
    Qvrc     : REAL := (5e-4)*(5e-4);   // RC-Prozessrauschen
    Rmeas    : REAL := (0.07)*(0.07); // Spannungs-Messrauschen

	(* Zwischenvariablen *)
    a_RC     : REAL;   // exp(-dt/(R1*C1))
    y_est    : REAL;
    innov    : REAL;
    S_pred   : REAL;
    K1, K2   : REAL;  // Kalman-Gain
    SOC_EKF  : REAL := 0.0;   // Ausgabe SoC in %
	
	// EKF-basierte SOC-Puffer (15 Sekunden Mittelung)
    SOC_EKF_Buffer        : ARRAY [0..59] OF REAL;   // Puffer für 15 letzte SOC-Werte
    Average_SOC_EKF       : REAL;                    // gemittelter SOC (EKF)
    EKF_BufferIndex       : INT := 0;
    EKF_BufferCount       : INT := 0;
	
	first_SOC_EKF 						: REAL := 0.0; 			// Erster Eintrag im Array SOC
	last_SOC_EKF 						: REAL := 0.0;			// Zu suchender letzter SoC-Wert, der nicht 0 ist
	
	tickCounter 			: INT := 0; // Zählt Durchläufe des Programms
	doEKF   			: BOOL := FALSE; // gibt immer nach 200 Durchläufen den EKF frei

	//Laufzeit/Ladezeitvorhersage
	Running_Time  					: REAL;					//Aktueller wert der Laufzeitvorhersage
	last_Running_Time				: REAL;					//Letzter wert der Laufzeitvorhersage
	Charging_Time 					: REAL; 				//Aktueller wert der Ladezeitvorhersage
	Charging_Time_Buffer			: ARRAY [0..119] OF REAL;
	Charging_Time_Look_Up_Table 	: ARRAY[0..100] OF REAL := [ 11826.0, 11710.8, 11592.0, 11476.8, 11361.6, 11246.4, 11131.2, 11012.4, 10893.6, 10778.4, 10659.6, 10540.8, 10422.0, 10303.2, 10184.4, 10065.6, 9943.2, 9820.8, 9698.4, 9572.4, 9446.4, 9320.4, 9194.4, 9068.4, 8938.8, 8809.2, 8679.6, 8550.0, 8416.8, 8283.6, 8150.4, 8017.2, 7884.0, 7747.2, 7610.4, 7473.6, 7336.8, 7196.4, 7056.0, 6915.6, 6775.2, 6634.8, 6490.8, 6346.8, 6202.8, 6055.2, 5907.6, 5760.0, 5612.4, 5461.2, 5310.0, 5158.8, 5007.6, 4852.8, 4698.0, 4543.2, 4384.8, 4226.4, 4064.4, 3902.4, 3740.4, 3578.4, 3412.8, 3247.2, 3081.6, 2912.4, 2743.2, 2574.0, 2401.2, 2228.4, 2055.6, 1882.8, 1706.4, 1530.0, 1353.6, 1173.6, 993.6, 813.6, 633.6, 450.0, 266.4, 82.8, 0.0, 0.0, 0.0, 0.0, 0.0, 0.0, 0.0, 0.0, 0.0, 0.0, 0.0, 0.0, 0.0, 0.0, 0.0, 0.0, 0.0, 0.0 ];
	
	
	// weiches Anfahren nach Laden
	wasCharging          : BOOL := FALSE;
    isCharging           : BOOL;
    ekfSoftStartCounter  : INT := 0;   // in Sekunden

	// Begrenzung des SOC Updates
	deltaSOC 	:REAL :=0;
	
	//x_Vrc clamping Variablen
	deltaVrc 	:REAL :=0;
    idx : INT;
    j   : INT;
	// Notfall Berechnung 
	CC_On :BOOL := FALSE;

	// reInit bei nicht logischen Werten
    socDeviationCounter : INT := 0;        // wie lange EKF von OCV-SOC abweicht
    socDeviationThreshold : INT := 5;     // 5 Sekunden Abweichung
    maxAllowedDeviation : REAL := 10;     // >10 % Abweichung → Verdacht Fehler
    socByVoltage : REAL;                   // SOC aus reiner OCV Schätzung
	idx_ocv      : INT :=0;					// merkt sich idx_min aus SOC lookup
	
END_VAR

//Notfalllberechnung 
//Wenn Einbrüche des SOC beim Konfiguration aktivieren oder Jobs schicken zu stark werden mit CCAn auf Coulomb Counting only umstellen
 CC_On := FALSE;  //TRUE für CC an

//Abschaltung SPS über den Shutdown Taster am Roboter selber
IF shutdownButton THEN
	shutdown(DELAY:=1, START:=TRUE);
END_IF

//Anpassung der Spannungs- und Stromwerte
batteryVoltage_V := (batteryVoltageRaw * scaleVoltage * 2.0)-(RobotData.factor_V_m*(batteryVoltageRaw * scaleVoltage * 2.0)+ RobotData.sum_V_b);
supplyCurrent_A :=  supplyCurrentRaw * 1000.0 / 270.0 / 32768 * 10 + RobotData.sum_I_b;

// SOC-Berechnung Anfang
// ab hier EKF Code 
tickCounter := tickCounter +1;
IF tickCounter >= 200 THEN 
	tickCounter :=0;
	doEKF := TRUE;
ELSE 
	doEKF := FALSE;
END_IF

I_Buffer[writeIndex] := supplyCurrent_A;
V_Buffer[writeIndex] := batteryVoltage_V;

//Index zyklisch weiterschieben
writeIndex := writeIndex + 1;
IF writeIndex >= 200 THEN
    writeIndex := 0;
END_IF
// EKF Code erstmal zu ende

// Wenn 200 Werte (~1min) geschrieben wurde
IF doEKF THEN
	// ab hier EKF
	// Berechung der mean Werte
	//korrektes Mitteln des Ringbuffers
	V_sum := 0;
	I_sum :=0;
	FOR j := 0 TO 199 DO
	    idx := writeIndex -1 - j;
	    IF idx < 0 THEN 
		idx := idx + 200; 
	    END_IF;
	    V_sum := V_sum + V_buffer[idx];
	    I_sum := I_sum + I_buffer[idx];
	END_FOR
	V_mean := V_sum / 200;
	I_mean := I_sum / 200;
	
	IF EKF_init  THEN
		OCV := V_mean + R0*I_mean + R1 * I_mean;  // SOC initialisieren mit erster Messung
		// Index mit kleinstem Abstand finden
		diff_min := ABS(OCV - OCV_Table[1]);  // Initialisierung mit erstem Wert 
		idx_min := 1;                         // Startindex 
		FOR i := 2 TO 201 DO
			diff := ABS(OCV - OCV_Table[i]);          // Abstand zum aktuellen Stützpunkt
			IF diff < diff_min THEN                   // Wenn Abstand kleiner als bisher 
				diff_min := diff;                     // neuen Minimalwert speichern 
				idx_min := i;                         // Index merken 
			END_IF
		END_FOR
		// SOC aus Tabelle übernehmen
		x_SOC := SOC_Table[idx_min]; // x_SOC initialisieren x_Vrc muss immer mit 0 initialisiert werden
		x_Vrc := 0;
		P11 := 1.0; 
		P22 := 1.0;   
    		P12 := 0.0; 
		P21 := 0.0;
		socDeviationCounter := 0;
	
		EKF_init := FALSE;  // Init Variable zurücksetzen
	END_IF
	
	// Berechnung der Ersatzschaltbild Parameter
	//clamping da nur für den Bereich 0.3-0.9 SOC gültig
	IF x_SOC <= 0.3 THEN 
		 param_SOC := 0.3;
	ELSIF x_SOC >= 0.9 THEN
		 param_SOC := 0.9;
	ELSE 
		param_SOC := x_SOC;
	END_IF
	R0 := 0.00903617*param_SOC*param_SOC - 0.00619734*param_SOC + 0.0861489;
    R1 := -0.0710499*param_SOC*param_SOC + 0.091486*param_SOC - 0.0118801;
    C1 := 4190.91*param_SOC*param_SOC - 5543.71*param_SOC + 2580.68;
	
	
	// weiches Anfahren nach dem Laden
	isCharging := (I_mean < 0);    // Schwellwert anpassen
	IF isCharging THEN
	    wasCharging := TRUE;
	ELSE
	    IF wasCharging THEN
	        // Gerade von Laden -> Entladen gewechselt
	        ekfSoftStartCounter := 10;   // z.B. 10s sanfter Übergang
	        wasCharging := FALSE;
	    END_IF
	END_IF
	// Dynamisches Messrauschen für sanften Übergang
	IF ekfSoftStartCounter > 0 THEN
	    Rmeas := 10.0 * (0.07)*(0.07);   // Spannung 10x weniger „glauben“
	    ekfSoftStartCounter := ekfSoftStartCounter - 1;
	ELSE
	    Rmeas := (0.07)*(0.07);;
	END_IF
	
	// 1) Vorhersage 
	// SOC_k+1 = SOC_k - dt*I/Q 
	x_SOC := x_SOC - (dt_ekf * I_mean) / Qbatt;
	IF x_SOC < 0 THEN 
		x_SOC := 0;
	ELSIF x_SOC > 1 THEN 
		x_SOC := 1;
	END_IF
	// Vrc_k+1 = exp(-dt/(R1*C1))*Vrc_k + R1*(1-exp(..))*I 
	a_RC := EXP( -dt_ekf / (R1 * C1) );
	x_Vrc := a_RC * x_Vrc + R1 * (1 - a_RC) * I_mean;
	
	IF I_mean > 0 AND (NOT CC_On) THEN  //Update nur während Entladung ansonsten nur Coulomb Counting	
		// Kovarianzmatrix P updaten (P = A*P*A' + Q) 
		P11 := P11 + Qz;                     // Unsicherheit im SOC wächst durch Modellrauschen
		P22 := (a_RC*a_RC)*P22 + Qvrc;       // Unsicherheit im RC-Zweig
		P12 := a_RC * P12;					 // Kreuzkovarianzen
		P21 := a_RC * P21;
		
		// 2) Messvorhersage mit LUT
		// Index mit kleinstem Abstand finden
		diff_min := ABS(x_SOC - SOC_Table[1]);  // Initialisierung mit erstem Wert 
		idx_min := 1;                         // Startindex 
		FOR i := 2 TO 201 DO
    		diff := ABS(x_SOC - SOC_Table[i]);          // Abstand zum aktuellen Stützpunkt
			IF diff < diff_min THEN                   // Wenn Abstand kleiner als bisher 
				diff_min := diff;                     // neuen Minimalwert speichern 
				idx_min := i;                         // Index merken
			END_IF
		END_FOR
		idx_ocv := idx_min; 		      // Index merken für ReInit		
		
		// OCV aus Tabelle übernehmen
		OCV := OCV_Table[idx_min];
		
		// dOCV/dSOC berechnen
		IF idx_min = 1 THEN
			(* Unterer Rand: nur obere Differenz verfügbar *)
			dVdSOC := (OCV_Table[2] - OCV_Table[1]) / (SOC_Table[2] - SOC_Table[1]);
		ELSIF idx_min = 201 THEN
			(* Oberer Rand: nur untere Differenz verfügbar *)
			dVdSOC := (OCV_Table[201] - OCV_Table[200]) / (SOC_Table[201] - SOC_Table[200]);
		ELSE
			(* Mittelwert aus oberer und unterer Differenz *)
			dVdSOC := ((OCV_Table[idx_min+1] - OCV_Table[idx_min-1]) /
					   (SOC_Table[idx_min+1] - SOC_Table[idx_min-1]));
		END_IF
		y_est := OCV - x_Vrc - R0*I_mean;
		
		// 3) Innovation 
		innov := V_mean - y_est;
	
		// 4) Innovations-Kovarianz  S = CPC' + R 
		// C = [dOCV ,  -1] 
		S_pred := dVdSOC*(P11*dVdSOC + P12*(-1)) + (-1)*(P21*dVdSOC + P22*(-1)) + Rmeas;
		
		// 5) Kalman-Gain 
		K1 := (P11*dVdSOC + P12*(-1)) / S_pred;   // für SOC
		K2 := (P21*dVdSOC + P22*(-1)) / S_pred;   // für Vrc
			
		deltaSOC := K1 * innov; 
		// dVrc Clamp auf 0.1V um Ausreißer klein zu halten
		deltaVrc := K2 * innov;
		IF deltaVrc > 0.1 THEN 
			deltaVrc := 0.1; 
		END_IF;
		IF deltaVrc < -0.1 THEN 
			deltaVrc := -0.1; 
		END_IF;

		// 6) Zustands-Update 
		x_SOC := x_SOC + deltaSOC;
		x_Vrc := x_Vrc + deltaVrc;
	
		IF x_SOC < 0 THEN x_SOC := 0;
		ELSIF x_SOC > 1 THEN x_SOC := 1;
		END_IF
		
		// 7) Kovarianz-Update P = (I - K*H)*P 
		P11 := P11 - K1*(dVdSOC*P11 + -1*P21);
		P12 := P12 - K1*(dVdSOC*P12 + -1*P22);
		P21 := P21 - K2*(dVdSOC*P11 + -1*P21);
		P22 := P22 - K2*(dVdSOC*P12 + -1*P22);
	END_IF
	
	// 8) Prozent-Ausgabe 
	SOC_EKF := x_SOC * 100.0;

	//ReInit falls SOC Springt 
	IF ABS(SOC_EKF - Average_SOC_EKF) > maxAllowedDeviation THEN
	    socDeviationCounter := socDeviationCounter + 1;
	ELSE
	    socDeviationCounter := 0;
	END_IF

	//ReInit Bedingungen
	IF (socDeviationCounter > socDeviationThreshold) AND (I_mean > 0) THEN 
	     EKF_init := TRUE;
	END_IF
	
	// EKF-SOC Mittelung über 60 s 
	SOC_EKF_Buffer[EKF_BufferIndex] := SOC_EKF;

	// Index erhöhen und ggf. zurücksetzen
	EKF_BufferIndex := EKF_BufferIndex + 1;
	IF EKF_BufferIndex >= 60 THEN
	    EKF_BufferIndex := 0;
	END_IF

	// BufferCount bis 60 erhöhen
	IF EKF_BufferCount < 60 THEN
	    EKF_BufferCount := EKF_BufferCount + 1;
	END_IF

	// Mittelwert berechnen
	Average_SOC_EKF := 0.0;
	FOR i := 0 TO (EKF_BufferCount - 1) DO
	    Average_SOC_EKF := Average_SOC_EKF + SOC_EKF_Buffer[i];
	END_FOR
	Average_SOC_EKF := Average_SOC_EKF / EKF_BufferCount;

	// Laufzeitberechnung basierend auf EKF-SOC
	IF I_mean > 0 AND EKF_BufferCount = 60 THEN
	    first_SOC_EKF := SOC_EKF_Buffer[0];
	    last_SOC_EKF  := SOC_EKF_Buffer[59];

	    IF last_SOC_EKF > 0 THEN
	        IF first_SOC_EKF > last_SOC_EKF + 0.05 THEN  // kleinerer Schwellwert evtl. sinnvoll
	            Running_Time := (Average_SOC_EKF / (first_SOC_EKF - last_SOC_EKF)) * EKF_BufferCount;
	            last_Running_Time := Running_Time;
	        ELSE
	            Running_Time := last_Running_Time;
 	       END_IF
 	   ELSE
	        Running_Time := 0.0;
 	   END_IF
	ELSE
	    Running_Time := 0.0;
	END_IF

	// Ladezeitberechnung (nur wenn Strom negativ)
	IF supplyCurrent_A < 0 THEN
	    Charging_Time := Charging_Time_Look_Up_Table[REAL_TO_INT(Average_SOC_EKF)];
	ELSE
	    Charging_Time := 0.0;
	END_IF
	// EKF ENDE
END_IF
//SOC-Berechnung Ende

//Sicherheitsabschaltung, wenn Roboterakku zu gering ( beim einstecken manchmal gibts einen Stromsprung bis 30A messfehelr wahrscheinlich)
// kann auf dem Roboter der mit Platine fährt auskommentiert werden!!!
IF batteryVoltage_V < 12 AND Average_SOC_EKF < 10 THEN   
	shutdownTrigger := TRUE;
END_IF

stMqtt_HAWino_IN.fActualBatteryVoltage := batteryVoltage_V;
stMqtt_HAWino_IN.fActualBatteryCurrent := supplyCurrent_A;
stMqtt_HAWino_IN.fSoC := Average_SOC_EKF;					
stMqtt_HAWino_IN.nEstimatedRunningTime := Running_Time;
stMqtt_HAWino_IN.nEstimatedChargingTime := Charging_Time;

END_PROGRAM

// ---- POUs/HAWinoCore/05_Bahnplanung/FB_CollisionAvoidance.TcPOU
FUNCTION_BLOCK FB_CollisionAvoidance
VAR_INPUT
    xrePosX        : REAL;
    xrePosY        : REAL;
    xreOwnAngle    : REAL;   (* aktueller Fahrwinkel in Grad *)
    xreOwnSpeed    : REAL;   (* aktuelle Eigengeschwindigkeit cm/s *)
    xreRobotX      : ARRAY[0..2] OF REAL;
    xreRobotY      : ARRAY[0..2] OF REAL;
    xboRobotActive : ARRAY[0..2] OF BOOL;
END_VAR
VAR_OUTPUT
    yreDynGx        : REAL;
    yreDynGy        : REAL;
    yboStop         : BOOL;
    yboWarning      : BOOL;
    yreMinDist      : REAL;
    yreSpeedFactor  : REAL;   (* 0.0..1.0 — Geschwindigkeitsskalierung *)
END_VAR
VAR
    _inIdx          : INT;
    _reDiffX        : REAL;
    _reDiffY        : REAL;
    _reDist         : REAL;
    _reDistSq       : REAL;
    _reRepulse      : REAL;
    _reWeight       : REAL;

    (* Winkel zwischen Fahrtrichtung und Verbindungslinie zum anderen Roboter *)
    _reAngleToRobot : REAL;   (* Winkel zur Verbindungslinie in Grad *)
    _reRelAngle     : REAL;   (* relativer Winkel zur Fahrtrichtung  *)
    _reAsymFactor   : REAL;   (* Asymmetriefaktor: links > rechts    *)
    _reFrontFactor  : REAL;   (* Verstärkung wenn Roboter frontal    *)

    (* Rechts-Bias: verschiebt Abstoßungsvektor leicht nach rechts *)
    _reOwnAngleRad  : REAL;
    _reRightX       : REAL;   (* Rechtsvektor des eigenen Roboters   *)
    _reRightY       : REAL;
    _reBiasX        : REAL;
    _reBiasY        : REAL;

    (* Geschwindigkeitsskalierung *)
    _reDynRepulseRad : REAL;
    _reDynRepulseK   : REAL;

    (* Basisparameter *)
    _creBaseRepulseK   : REAL := 1000.0;
    _creBaseRepulseRad : REAL := 60.0; //60
    _creWarnDist       : REAL := 100.0;
    _creStopDist       : REAL := 18.0;
    _creMaxSpeed       : REAL := 80.0;    (* Maximalgeschwindigkeit cm/s *)

    (* Asymmetrie *)
    _creRightBias      : REAL := 0.01;    (* Stärke des Rechtsversatzes 0..1 *)
    _creFrontThreshold : REAL := 50.0;    (* Winkel ab dem "frontal" gilt    *)
    _creFrontBoost     : REAL := 10;     (* Verstärkung bei frontalem Kurs  *)

    (* Geschwindigkeitsskalierung *)
    _creSpeedScaleK    : REAL := 1.5;     (* max. Skalierungsfaktor Kraft    *)
    _creSpeedScaleRad  : REAL := 1.8;     (* max. Skalierungsfaktor Radius   *)

    (* Geschwindigkeitsreduktion *)
    _creSlowDist       : REAL := 75.0;    (* ab hier verlangsamen            *)
    _creStopDist2      : REAL := 18.0;    (* Vollstopp                       *)
END_VAR

(* ── Reset ─────────────────────────────────────────── *)
yreDynGx        := 0.0;
yreDynGy        := 0.0;
yboStop         := FALSE;
yboWarning      := FALSE;
yreMinDist      := _creBaseRepulseRad * _creSpeedScaleRad;
yreSpeedFactor  := 1.0;

(* ── Geschwindigkeitsabhängige Parameter ───────────── *)
(* Normierte Eigengeschwindigkeit 0..1 *)
_reWeight := MIN(xreOwnSpeed / _creMaxSpeed, 1.0);

(* Wirkradius wächst linear mit Geschwindigkeit *)
_reDynRepulseRad := _creBaseRepulseRad *
                    (1.0 + _reWeight * (_creSpeedScaleRad - 1.0));

(* Abstoßungskraft wächst linear mit Geschwindigkeit *)
_reDynRepulseK   := _creBaseRepulseK *
                    (1.0 + _reWeight * (_creSpeedScaleK - 1.0));

(* ── Rechtsvektor berechnen ────────────────────────── *)
(* 90° im Uhrzeigersinn = rechts relativ zur Fahrtrichtung *)
_reOwnAngleRad := xreOwnAngle * 3.14159265 / 180.0;
_reRightX      :=  SIN(_reOwnAngleRad);   (*  sin gibt rechts *)
_reRightY      := -COS(_reOwnAngleRad);   (* -cos gibt rechts *)

FOR _inIdx := 0 TO 2 DO
    IF NOT xboRobotActive[_inIdx] THEN CONTINUE; END_IF

    (* ── Abstand berechnen ─────────────────────────── *)
    _reDiffX := xrePosX - xreRobotX[_inIdx];
    _reDiffY := xrePosY - xreRobotY[_inIdx];
    _reDist  := SQRT(_reDiffX * _reDiffX + _reDiffY * _reDiffY);

    IF _reDist < yreMinDist THEN
        yreMinDist := _reDist;
    END_IF

    (* ── Zonen ─────────────────────────────────────── *)
    IF _reDist < _creStopDist THEN
        yboStop := TRUE;
    END_IF

    IF _reDist < _creWarnDist THEN
        yboWarning := TRUE;
    END_IF

    (* ── Geschwindigkeitsreduktion ─────────────────── *)
    (* Stufenlose Reduktion zwischen SlowDist und StopDist *)
    IF _reDist < _reDynRepulseRad THEN
        IF _reDist <= _creStopDist2 THEN
            yreSpeedFactor := 0.0;
        ELSIF _reDist < _creSlowDist THEN
            yreSpeedFactor := MIN(yreSpeedFactor,
                                  (_reDist - _creStopDist2) /
                                  (_creSlowDist - _creStopDist2));
        END_IF
    END_IF

    IF _reDist > _reDynRepulseRad THEN CONTINUE; END_IF
    IF _reDist < 0.1 THEN CONTINUE; END_IF

    (* ── Frontaler Kurs erkennen ───────────────────── *)
    (* Winkel zwischen Fahrtrichtung und Verbindungslinie *)
    _reAngleToRobot := FC_ATAN2(
                         xreY := -_reDiffY,
                         xreX := -_reDiffX)
                       * 180.0 / 3.14159265;

    _reRelAngle := _reAngleToRobot - xreOwnAngle;

    (* Auf [-180, +180] normieren *)
    WHILE _reRelAngle > 180.0  DO _reRelAngle := _reRelAngle - 360.0; END_WHILE
    WHILE _reRelAngle < -180.0 DO _reRelAngle := _reRelAngle + 360.0; END_WHILE

    (* Frontaler Kurs: anderer Roboter ist direkt vor uns *)
    IF ABS(_reRelAngle) < _creFrontThreshold THEN
        _reFrontFactor := _creFrontBoost *
                          (1.0 - ABS(_reRelAngle) / _creFrontThreshold);
    ELSE
        _reFrontFactor := 1.0;
    END_IF

    (* ── Asymmetriefaktor berechnen ────────────────── *)
    (* Skalarprodukt mit Rechtsvektor:
       > 0 = anderer Roboter ist rechts von uns → weniger abstoßen
       < 0 = anderer Roboter ist links von uns  → mehr abstoßen
       → Roboter weicht nach rechts aus                          *)
    _reAsymFactor := 1.0 - _creRightBias *
                     (_reDiffX * _reRightX + _reDiffY * _reRightY) /
                     _reDist;

    (* ── Abstoßungsstärke ──────────────────────────── *)
    _reDistSq  := MAX(_reDist * _reDist, 1.0);
    _reRepulse := _reDynRepulseK / _reDistSq
                  * _reAsymFactor
                  * _reFrontFactor;

    (* Zusätzliche Verstärkung im Warnbereich *)
    IF _reDist < _creWarnDist THEN
        _reRepulse := _reRepulse *
                      (1.0 + (_creWarnDist - _reDist) /
                              _creWarnDist * 2.0);
    END_IF

    (* ── Rechts-Bias zum Abstoßungsvektor addieren ─── *)
    (* Verschiebt den Vektor leicht nach rechts damit
       der Roboter eine Rechtskurve bevorzugt           *)
    _reBiasX := _reRightX * _creRightBias * _reRepulse * 0.3;
    _reBiasY := _reRightY * _creRightBias * _reRepulse * 0.3;

    yreDynGx := yreDynGx + _reRepulse * _reDiffX / _reDist + _reBiasX;
    yreDynGy := yreDynGy + _reRepulse * _reDiffY / _reDist + _reBiasY;

END_FOR

(* SpeedFactor auf 0 erzwingen bei Stopp *)
IF yboStop THEN
    yreSpeedFactor := 0.0;
END_IF

END_FUNCTION_BLOCK

// ---- POUs/HAWinoCore/05_Bahnplanung/FB_CollisionAvoidanceV2.TcPOU
FUNCTION_BLOCK FB_CollisionAvoidanceV2
VAR_INPUT
    xrePosX        : REAL;
    xrePosY        : REAL;
    xreOwnAngle    : REAL;   (* aktueller Fahrwinkel in Grad *)
    xreOwnSpeed    : REAL;   (* Eigengeschwindigkeit in cm/s *)
    xreRobotX      : ARRAY[0..2] OF REAL;
    xreRobotY      : ARRAY[0..2] OF REAL;
    xboRobotActive : ARRAY[0..2] OF BOOL;
END_VAR
VAR_OUTPUT
    yreDynGx           : REAL;   (* Abstoßungsvektor X — Weltkoordinaten *)
    yreDynGy           : REAL;   (* Abstoßungsvektor Y — Weltkoordinaten *)
    yboStop            : BOOL;
    yboWarning         : BOOL;
    yreMinDist         : REAL;   (* kleinster Abstand zu einem Roboter   *)
    yreSpeedFactor     : REAL;   (* 0.0..1.0 Geschwindigkeitsskalierung  *)
    yreNearestRobotDir : REAL;   (* Richtung zum nächsten Roboter in Grad *)
END_VAR
VAR
    _inIdx          : INT;

    (* Abstandsvektor in Weltkoordinaten *)
    _reDiffX        : REAL;   (* zeigt VON fremd ZU uns *)
    _reDiffY        : REAL;
    _reDist         : REAL;

    (* Eigene Fahrtrichtung *)
    _reOwnRad       : REAL;
    _reFwdX         : REAL;   (* Einheitsvektor vorwärts *)
    _reFwdY         : REAL;
    _reRightX       : REAL;   (* Einheitsvektor rechts   *)
    _reRightY       : REAL;

    (* Lokale Koordinaten: Projektion auf Fwd/Right *)
    _reLong         : REAL;   (* > 0 = Roboter vor uns   *)
    _reLat          : REAL;   (* > 0 = Roboter rechts    *)

    (* Ellipse *)
    _reRadFwd       : REAL;   (* aktueller Vorwärtsradius *)
    _reRadLat       : REAL;   (* aktueller Seitwärtsradius *)
    _reEllipse      : REAL;   (* 0=Mitte, 1=Rand, >1=außen *)

    (* Kraft in lokalen Koordinaten *)
    _reForceLong    : REAL;   (* Kraft in Längsrichtung  *)
    _reForceLat     : REAL;   (* Kraft in Querrichtung   *)
    _reForceBase    : REAL;   (* Basiskraft              *)
    _reSoftFactor   : REAL;   (* Weicher Einstieg 0..1   *)
    _reFrontBoost   : REAL;   (* Frontalverstärkung      *)
    _reAsym         : REAL;   (* Asymmetriefaktor        *)

    (* Hilfsvariable für nächsten Roboter *)
    _reNearestDist  : REAL;

    (* Geschwindigkeit normiert 0..1 *)
    _reSpeedNorm    : REAL;

    (* ── Tuning-Parameter ────────────────────────── *)

    (* Wirkzone *)
    _creBaseRadFwd  : REAL := 200.0;   //150(* Vorwärtsradius bei Stillstand cm  *)
    _creBaseRadLat  : REAL := 60.0;   (* Seitwärtsradius bei Stillstand cm *) //80

    (* Geschwindigkeitsskalierung *)
    _creMaxSpeed    : REAL := 80.0;   (* Maximalgeschwindigkeit cm/s       *)
    _creScaleRadFwd : REAL := 3.0;    (* Faktor Vorwärtsradius bei Vmax    *)
    _creScaleRadLat : REAL := 1.0;    (* Faktor Seitwärtsradius bei Vmax   *)
    _creScaleK      : REAL := 1.8;    (* Faktor Kraft bei Vmax             *)

    (* Kraft *)
    _creBaseK       : REAL := 1800.0;  (* Basiskraft                        *)

    (* Weicher Einstieg *)
    (* 0 = linear ab Rand, 1 = sehr weich, erst in der Mitte stark *)
    _creSoftness    : REAL := 0.1;

    (* Frontalverstärkung *)
    (* Wie viel stärker wird abgestoßen wenn Roboter direkt vor uns *)
    _creFrontBoost  : REAL := 5.0;
    (* Öffnungswinkel für "frontal" in Grad *)
    _creFrontAngle  : REAL := 30.0;

    (* Rechts-Bias *)
    (* Anteil der Kraft der seitlich nach rechts verschoben wird *)
    _creRightBias   : REAL := 0.1;

    (* Zonengrenzen *)
    _creWarnDist    : REAL := 38.0;
    _creStopDist    : REAL := 18.0;
    _creSlowDist    : REAL := 60.0;//50
END_VAR


(* ════════════════════════════════════════════════════
   INITIALISIERUNG
   ════════════════════════════════════════════════════ *)
yreDynGx           := 0.0;
yreDynGy           := 0.0;
yboStop            := FALSE;
yboWarning         := FALSE;
yreMinDist         := 9999.0;
yreSpeedFactor     := 1.0;
yreNearestRobotDir := 0.0;
_reNearestDist     := 9999.0;

(* ── Eigene Fahrtrichtung in Einheitsvektoren ───────── *)
_reOwnRad  := xreOwnAngle * 3.14159265 / 180.0;
_reFwdX    :=  COS(_reOwnRad);
_reFwdY    :=  SIN(_reOwnRad);
_reRightX  :=  SIN(_reOwnRad);    (* 90° im Uhrzeigersinn *)
_reRightY  := -COS(_reOwnRad);

(* ── Geschwindigkeit normieren ──────────────────────── *)
_reSpeedNorm := MIN(xreOwnSpeed / _creMaxSpeed, 1.0);

(* ── Dynamische Wirkzone ────────────────────────────── *)
_reRadFwd := _creBaseRadFwd *
             (1.0 + _reSpeedNorm * (_creScaleRadFwd - 1.0));
_reRadLat := _creBaseRadLat *
             (1.0 + _reSpeedNorm * (_creScaleRadLat - 1.0));

(* ════════════════════════════════════════════════════
   HAUPTSCHLEIFE
   ════════════════════════════════════════════════════ *)
FOR _inIdx := 0 TO 2 DO
    IF NOT xboRobotActive[_inIdx] THEN CONTINUE; END_IF

    (* ── Abstandsvektor ────────────────────────────── *)
    _reDiffX := xrePosX - xreRobotX[_inIdx];
    _reDiffY := xrePosY - xreRobotY[_inIdx];
    _reDist  := SQRT(_reDiffX * _reDiffX + _reDiffY * _reDiffY);

    IF _reDist < 0.1 THEN CONTINUE; END_IF

    (* ── Nächsten Roboter tracken ───────────────────── *)
    IF _reDist < _reNearestDist THEN
        _reNearestDist     := _reDist;
        yreMinDist         := _reDist;
        (* Richtung ZUM anderen Roboter: -Diff *)
        yreNearestRobotDir := FC_ATAN2(
                                xreY := -_reDiffY,
                                xreX := -_reDiffX)
                              * 180.0 / 3.14159265;
    END_IF

    (* ── Projektion auf lokale Achsen ──────────────── *)
    (* _reDiff zeigt von fremd zu uns — für Projektion  *)
    (* "wo ist der andere" umkehren: von uns zu fremd   *)
    _reLong := -(_reDiffX * _reFwdX   + _reDiffY * _reFwdY);
    _reLat  := -(_reDiffX * _reRightX + _reDiffY * _reRightY);

    (* ── Ellipsenwert berechnen ─────────────────────── *)
    IF _reLong >= 0.0 THEN
        (* Vor uns: voller Radius *)
        _reEllipse :=
            (_reLong / _reRadFwd) * (_reLong / _reRadFwd) +
            (_reLat  / _reRadLat) * (_reLat  / _reRadLat);
    ELSE
        (* Hinter uns: stark reduzierter Radius *)
        _reEllipse :=
            (_reLong / (_reRadFwd * 0.3)) * (_reLong / (_reRadFwd * 0.3)) +
            (_reLat  / (_reRadLat * 0.5)) * (_reLat  / (_reRadLat * 0.5));
    END_IF

    (* Außerhalb: kein Einfluss *)
    IF _reEllipse > 1.0 THEN CONTINUE; END_IF

    (* ── Zonen prüfen ───────────────────────────────── *)
    IF _reDist < _creStopDist THEN
        yboStop := TRUE;
    END_IF
    IF _reDist < _creWarnDist THEN
        yboWarning := TRUE;
    END_IF

    (* ── Geschwindigkeitsreduktion ─────────────────── *)
    IF _reDist < _creSlowDist THEN
        IF _reDist <= _creStopDist THEN
            yreSpeedFactor := 0.0;
        ELSE
            yreSpeedFactor := MIN(
                yreSpeedFactor,
                (_reDist - _creStopDist) / (_creSlowDist - _creStopDist));
        END_IF
    END_IF

    (* ════════════════════════════════════════════════
       KRAFT IN LOKALEN KOORDINATEN BERECHNEN
       ════════════════════════════════════════════════ *)

    (* ── Basiskraft: quadratisch abfallend ──────────── *)
    _reForceBase := _creBaseK *
                    (1.0 + _reSpeedNorm * (_creScaleK - 1.0)) /
                    MAX(_reDist * _reDist, 1.0);

    (* ── Weicher Einstieg ───────────────────────────── *)
    (* Am Rand der Ellipse (=1): Faktor nahe 0           *)
    (* In der Mitte (=0): Faktor = 1                     *)
    (* _creSoftness steuert wie schnell der Anstieg ist  *)
    _reSoftFactor := (1.0 - _reEllipse) /
                     (1.0 - _reEllipse + _creSoftness);

    _reForceBase := _reForceBase * _reSoftFactor;

    (* ── Frontalverstärkung ─────────────────────────── *)
    (* Wenn _reLong >> _reLat: anderer Roboter fast direkt vor uns *)
    IF _reLong > 0.0 THEN
        _reFrontBoost := 1.0 + (_creFrontBoost - 1.0) *
                         MAX(0.0,
                             1.0 - ABS(_reLat) /
                             (_reLong * TAN(_creFrontAngle *
                                           3.14159265 / 180.0)
                              + 0.001));
    ELSE
        _reFrontBoost := 1.0;
    END_IF

    _reForceBase := _reForceBase * _reFrontBoost;

    (* ── Kraft aufteilen in Längs- und Querkomponente ── *)
    (* Längskomponente: direkt vom anderen Roboter weg    *)
    (* Querkomponente:  seitlich ausweichen mit Bias      *)

    (* Längsanteil: proportional zur Längsprojektion *)
    _reForceLong := _reForceBase * _reLong / MAX(_reDist, 1.0);

    (* Queranteil: proportional zur Lateralprojektion
       + Rechts-Bias: konstante Komponente nach rechts   *)
    _reForceLat  := _reForceBase * _reLat / MAX(_reDist, 1.0);

    (* ── Asymmetrie: Rechts-Bias ────────────────────── *)
    (* Roboter links  (_reLat < 0): stärker nach rechts  *)
    (* Roboter rechts (_reLat > 0): schwächer ausweichen *)
    _reAsym := 1.0 + _creRightBias * (-_reLat / MAX(_reDist, 1.0));
    _reAsym := MAX(0.2, MIN(_reAsym, 2.5));

    (* Rechts-Bias: feste Querkomponente nach rechts addieren *)
    _reForceLat := _reForceLat +
                   _creRightBias * _reForceBase * _reAsym;

    (* ════════════════════════════════════════════════
       ZURÜCK IN WELTKOORDINATEN
       ════════════════════════════════════════════════ *)
    (* Längsanteil entlang -Fwd (von anderem Roboter weg) *)
    (* Queranteil entlang +Right (nach rechts ausweichen) *)
    yreDynGx := yreDynGx
                - _reForceLong * _reFwdX      (* Längs: weg vom Roboter  *)
                + _reForceLat  * _reRightX;   (* Quer:  nach rechts      *)

    yreDynGy := yreDynGy
                - _reForceLong * _reFwdY
                + _reForceLat  * _reRightY;

END_FOR

IF yboStop THEN
    yreSpeedFactor := 0.0;
END_IF

END_FUNCTION_BLOCK

// ---- POUs/HAWinoCore/05_Bahnplanung/FB_CollisionAvoidanceV22.TcPOU
FUNCTION_BLOCK FB_CollisionAvoidanceV22
VAR_INPUT
    xrePosX        : REAL;
    xrePosY        : REAL;
    xreOwnAngle    : REAL;
    xreOwnSpeed    : REAL;
    xreRobotX      : ARRAY[0..2] OF REAL;
    xreRobotY      : ARRAY[0..2] OF REAL;
    xboRobotActive : ARRAY[0..2] OF BOOL;
END_VAR
VAR_OUTPUT
    yreDynGx           : REAL;
    yreDynGy           : REAL;
    yboStop            : BOOL;
    yboWarning         : BOOL;
    yreMinDist         : REAL;
    yreSpeedFactor     : REAL;
    yreNearestRobotDir : REAL;
	yreAusgangsTest : REAL;
END_VAR
VAR
    _inIdx         : INT;
    _reDiffX       : REAL;
    _reDiffY       : REAL;
    _reDist        : REAL;
    _reRepulse     : REAL;
    _reNearestDist : REAL;

    (* Lokale Koordinaten für Bias *)
    _reOwnRad      : REAL;
    _reFwdX        : REAL;
    _reFwdY        : REAL;
    _reRightX      : REAL;
    _reRightY      : REAL;
    _reLong        : REAL;
    _reLat         : REAL;

    (* ── Tuning — nur diese 6 Parameter ───────────── *)
  //  _creRepulseRad  : REAL := 50.0;   (* Wirkradius in cm                  *) //70  alt aber weit entfernt    50 ziemlich dicht aber langsam
  //  _creRepulseK    : REAL := 3000.0; (* Abstoßungskraft                   *)
    _creStopDist    : REAL := 20.0;   (* Notstopp in cm                    *)
    _creWarnDist    : REAL := 45.0;   (* Warnung in cm                     *) //macht glaube nichts ???
    _creSlowDist    : REAL := 50.0;   (* Abbremsen ab hier                 *) // 80
    _creRightBias   : REAL := 0.0;   (* Rechtsversatz 0=kein Bias, 1=viel *)
	(* Wirkzone: Ellipse statt Kreis *)
_creRadFwd  : REAL := 80.0;   (* Vorwärtsradius — bestimmt Frühzeitigkeit *)
_creRadLat  : REAL := 40.0;    (* Seitwärtsradius — bestimmt seitlichen Abstand *)
_creRepulseK : REAL := 3000.0;
_reEllipse : REAL;
END_VAR

(* ── Reset ─────────────────────────────────────────── *)
yreDynGx           := 0.0;
yreDynGy           := 0.0;
yboStop            := FALSE;
yboWarning         := FALSE;
yreMinDist         := 9999.0;
yreSpeedFactor     := 1.0;
yreNearestRobotDir := 0.0;
_reNearestDist     := 9999.0;

(* ── Fahrtrichtung ──────────────────────────────────── *)
_reOwnRad := xreOwnAngle * 3.14159265 / 180.0;
_reFwdX   :=  COS(_reOwnRad);
_reFwdY   :=  SIN(_reOwnRad);
_reRightX :=  SIN(_reOwnRad);
_reRightY := -COS(_reOwnRad);

FOR _inIdx := 0 TO 2 DO
    IF NOT xboRobotActive[_inIdx] THEN CONTINUE; END_IF

    (* ── Abstand ───────────────────────────────────── *)
    _reDiffX := xrePosX - xreRobotX[_inIdx];
    _reDiffY := xrePosY - xreRobotY[_inIdx];
    _reDist  := SQRT(_reDiffX * _reDiffX + _reDiffY * _reDiffY);

    IF _reDist < 0.1 THEN CONTINUE; END_IF

    (* ── Nächsten Roboter ───────────────────────────── *)
    IF _reDist < _reNearestDist THEN
        _reNearestDist     := _reDist;
        yreMinDist         := _reDist;
        yreNearestRobotDir := FC_ATAN2(
                                xreY := -_reDiffY,
                                xreX := -_reDiffX)
                              * 180.0 / 3.14159265;
    END_IF

    (* ── Zonen ─────────────────────────────────────── *)
    IF _reDist < _creStopDist  THEN yboStop    := TRUE; END_IF
    IF _reDist < _creWarnDist  THEN yboWarning := TRUE; END_IF

    (* ── Geschwindigkeitsreduktion ─────────────────── *)
    IF _reDist < _creSlowDist THEN
        IF _reDist <= _creStopDist THEN
            yreSpeedFactor := 0.0;
        ELSE
            yreSpeedFactor := MIN(
                yreSpeedFactor,
                (_reDist - _creStopDist) /
                ( 1.15 * _creSlowDist - _creStopDist));
        END_IF
    END_IF

    (* ── Außerhalb Wirkradius ───────────────────────── *)
//     IF _reDist > _creRepulseRad THEN CONTINUE; END_IF
// 
//     (* ── Projektion ─────────────────────────────────── *)
   _reLong := -(_reDiffX * _reFwdX   + _reDiffY * _reFwdY);
    _reLat  := -(_reDiffX * _reRightX + _reDiffY * _reRightY);
// 
//     (* ── Nur reagieren wenn Roboter vor uns ist ─────── *)
//     (* Hinter uns: halbe Kraft                           *)
//     IF _reLong < 0.0 THEN
//         _reRepulse := (_creRepulseK / MAX(_reDist * _reDist, 1.0)) * 0.5;
//     ELSE
//         _reRepulse := _creRepulseK / MAX(_reDist * _reDist, 1.0) ;
//     END_IF
(* NEU — elliptisch: *)
IF _reLong >= 0.0 THEN
    _reEllipse := (_reLong / _creRadFwd) * (_reLong / _creRadFwd)
                + (_reLat  / _creRadLat) * (_reLat  / _creRadLat);
ELSE
    _reEllipse := (_reLong / (_creRadFwd * 0.3)) * (_reLong / (_creRadFwd * 0.3))
                + (_reLat  / (_creRadLat * 0.3)) * (_reLat  / (_creRadLat * 0.3));
END_IF

IF _reEllipse > 1.0 THEN CONTINUE; END_IF

(* Kraft bleibt wie bisher — basierend auf echtem Abstand *)
_reRepulse := _creRepulseK / MAX(_reDist * _reDist, 1.0);

    (* ── Geschwindigkeit skaliert Kraft ─────────────── *)
    _reRepulse := MAX(_reRepulse *
                  (1.0 + (xreOwnSpeed / 80.0) * 0.8), 1.2);

				  
    (* ── Abstoßungsvektor in Weltkoordinaten ────────── *)
    (* Direkte Abstoßung: weg vom anderen Roboter        *)
    yreDynGx := yreDynGx + _reRepulse * _reDiffX / _reDist;
    yreDynGy := yreDynGy + _reRepulse * _reDiffY / _reDist;

    (* ── Rechts-Bias: feste Komponente nach rechts ──── *)
    (* Nur wenn Roboter vor uns (_reLong > 0)            *)
    (* Stärker wenn Roboter links (_reLat < 0)           *)
    IF _reLong > 0.0 THEN
        yreDynGx := yreDynGx + _reRightX * _reRepulse * _creRightBias
                    * MAX(0.0, 1.0 - _reLat / MAX(_reDist, 1.0));
        yreDynGy := yreDynGy + _reRightY * _reRepulse * _creRightBias
                    * MAX(0.0, 1.0 - _reLat / MAX(_reDist, 1.0));
    END_IF

END_FOR

yreAusgangsTest := _reRepulse;

IF yboStop THEN yreSpeedFactor := 0.0; END_IF

END_FUNCTION_BLOCK

// ---- POUs/HAWinoCore/05_Bahnplanung/FB_CollisionAvoidanceV3_4.TcPOU
FUNCTION_BLOCK FB_CollisionAvoidanceV3_4
VAR_INPUT
    xrePosX        : REAL;
    xrePosY        : REAL;
    xreOwnAngle    : REAL;
    xreOwnSpeed    : REAL;
    xreRobotX      : ARRAY[0..2] OF REAL;
    xreRobotY      : ARRAY[0..2] OF REAL;
    xboRobotActive : ARRAY[0..2] OF BOOL;
	xinOwnID : INT;
END_VAR
VAR_OUTPUT
    yreDynGx           : REAL;
    yreDynGy           : REAL;
    yboStop            : BOOL;
    yboWarning         : BOOL;
    yreMinDist         : REAL;
    yreSpeedFactor     : REAL;
    yreNearestRobotDir : REAL;
	yreAusgangsTest : REAL;
END_VAR
VAR
    _inIdx         : INT;
    _reDiffX       : REAL;
    _reDiffY       : REAL;
    _reDist        : REAL;
    _reRepulse     : REAL;
    _reNearestDist : REAL;
	
	
	rToleranz        : REAL := 5.0; (* Dein "Bereich", z.B. 5 Grad *)
    rDifferenz       : REAL;
    bImBereich       : BOOL;
	
	
	_reToOtherX   : REAL;
_reToOtherY   : REAL;
	_reCross      : REAL;
_reFrontal    : REAL;
_rePerpX      : REAL;
_rePerpY      : REAL;
_rePerpWeight : REAL;
_aboPerpActive : ARRAY[0..2] OF BOOL;   (* Latch pro Roboter *)

    (* Lokale Koordinaten für Bias *)
    _reOwnRad      : REAL;
    _reFwdX        : REAL;
    _reFwdY        : REAL;
    _reRightX      : REAL;
    _reRightY      : REAL;
    _reLong        : REAL;
    _reLat         : REAL;

    (* ── Tuning — nur diese 6 Parameter ───────────── *)
    _creRepulseRad  : REAL := 60.0;   (* Wirkradius in cm                  *) //70  alt aber weit entfernt    50 ziemlich dicht aber langsam
    _creRepulseK    : REAL := 3000.0; (* Abstoßungskraft                   *)
    _creStopDist    : REAL := 20.0;   (* Notstopp in cm                    *)
    _creWarnDist    : REAL := 45.0;   (* Warnung in cm                     *) //macht glaube nichts ???
    _creSlowDist    : REAL := 100.0;   (* Abbremsen ab hier                 *)
    _creRightBias   : REAL := 1.5;   (* Rechtsversatz 0=kein Bias, 1=viel *)

END_VAR

(* ── Reset ─────────────────────────────────────────── *)
yreDynGx           := 0.0;
yreDynGy           := 0.0;
yboStop            := FALSE;
yboWarning         := FALSE;
yreMinDist         := 9999.0;
yreSpeedFactor     := 1.0;
yreNearestRobotDir := 0.0;
_reNearestDist     := 9999.0;

(* ── Fahrtrichtung ──────────────────────────────────── *)
_reOwnRad := xreOwnAngle * 3.14159265 / 180.0;
_reFwdX   :=  COS(_reOwnRad);
_reFwdY   :=  SIN(_reOwnRad);
_reRightX :=  SIN(_reOwnRad);
_reRightY := -COS(_reOwnRad);

FOR _inIdx := 0 TO 2 DO
    IF NOT xboRobotActive[_inIdx] THEN CONTINUE; END_IF

    (* ── Abstand ───────────────────────────────────── *)
    _reDiffX := xrePosX - xreRobotX[_inIdx];
    _reDiffY := xrePosY - xreRobotY[_inIdx];
    _reDist  := SQRT(_reDiffX * _reDiffX + _reDiffY * _reDiffY);

    IF _reDist < 0.1 THEN CONTINUE; END_IF

    (* ── Nächsten Roboter ───────────────────────────── *)
    IF _reDist < _reNearestDist THEN
        _reNearestDist     := _reDist;
        yreMinDist         := _reDist;
        yreNearestRobotDir := FC_ATAN2(
                                xreY := -_reDiffY,
                                xreX := -_reDiffX)
                              * 180.0 / 3.14159265;
    END_IF

    (* ── Zonen ─────────────────────────────────────── *)
    IF _reDist < _creStopDist  THEN yboStop    := TRUE; END_IF
    IF _reDist < _creWarnDist  THEN yboWarning := TRUE; END_IF

    (* ── Geschwindigkeitsreduktion ─────────────────── *)
    IF _reDist < _creSlowDist THEN
        IF _reDist <= _creStopDist THEN
            yreSpeedFactor := 0.0;
        ELSE
            yreSpeedFactor := MIN(
                yreSpeedFactor,
                (_reDist - _creStopDist) /
                (1 * _creSlowDist - _creStopDist));
        END_IF
    END_IF

    (* ── Latch-Reset: erst wenn deutlich außerhalb Wirkradius ── *)
    IF _reDist > _creRepulseRad * 1.5 THEN
        _aboPerpActive[_inIdx] := FALSE;
    END_IF

    (* ── Außerhalb Wirkradius: kein Repulse ─────────── *)
    IF _reDist > _creRepulseRad THEN CONTINUE; END_IF

    (* ── Projektion auf Fahrtrichtung ───────────────── *)
    _reLong := -(_reDiffX * _reFwdX   + _reDiffY * _reFwdY);
    _reLat  := -(_reDiffX * _reRightX + _reDiffY * _reRightY);

    (* ── Abstoßungskraft ────────────────────────────── *)
    IF _reLong < 0.0 THEN
        _reRepulse := (_creRepulseK / MAX(_reDist * _reDist, 1.0)) * 0.5;
    ELSE
        _reRepulse := _creRepulseK / MAX(_reDist * _reDist, 1.0);
    END_IF

    (* ── Geschwindigkeit skaliert Kraft ─────────────── *)
    _reRepulse := MAX(_reRepulse *
                  (1.0 + (xreOwnSpeed / 80.0) * 0.8), 1.2);

    (* ── Abstoßungsvektor in Weltkoordinaten ────────── *)
    yreDynGx := yreDynGx + _reRepulse * _reDiffX / _reDist;
    yreDynGy := yreDynGy + _reRepulse * _reDiffY / _reDist;

    (* ══════════════════════════════════════════════════
       SEITLICHE ABLENKUNG MIT HYSTERESE-LATCH
       SET:   Roboter ist vor uns (_reLong > 0)
       AKTIV: solange Latch gesetzt, unabhängig von _reLong
       RESET: erst wenn Abstand > _creRepulseRad * 1.5
       ══════════════════════════════════════════════════ *)

    (* SET: Roboter erkennbar vor uns *)
    IF _reLong > 0.0 THEN
        _aboPerpActive[_inIdx] := TRUE;
    END_IF

    IF _aboPerpActive[_inIdx] THEN

        (* Einheitsvektoren: Richtung vom eigenen Roboter zum anderen *)
        _reToOtherX := -_reDiffX / _reDist;
        _reToOtherY := -_reDiffY / _reDist;

        (* Kreuzprodukt Z: eigener Fahrvektor × Richtung-zum-anderen  *)
        (* > 0: anderer Roboter rechts  -> wir weichen links aus       *)
        (* < 0: anderer Roboter links   -> wir weichen rechts aus      *)
        _reCross := _reFwdX * _reToOtherY - _reFwdY * _reToOtherX;

        (* Wie frontal ist die Begegnung?                              *)
        (* 1.0 = exakt frontal, 0.0 = seitlich vorbei                 *)
        _reFrontal := _reFwdX * _reToOtherX + _reFwdY * _reToOtherY;
        _reFrontal := MAX(0.0, _reFrontal);

        (* Senkrechter Vektor, Richtung per Kreuzprodukt               *)
        (* Tiebreaker per RoboterID bei exakt symmetrischem Frontalfall*)
        IF ABS(_reCross) < 0.15 THEN
            (* Exakt frontal: ID-basierte feste Seite -> kein Deadlock *)
            IF xinOwnID MOD 2 = 0 THEN
                _rePerpX :=  _reToOtherY;
                _rePerpY := -_reToOtherX;
            ELSE
                _rePerpX := -_reToOtherY;
                _rePerpY :=  _reToOtherX;
            END_IF
        ELSIF _reCross >= 0.0 THEN
            (* Anderer rechts -> links ausweichen *)
            _rePerpX := -_reToOtherY;
            _rePerpY :=  _reToOtherX;
        ELSE
            (* Anderer links -> rechts ausweichen *)
            _rePerpX :=  _reToOtherY;
            _rePerpY := -_reToOtherX;
        END_IF

        (* Gewichtung: je frontaler, desto stärker der Perp-Anteil    *)
        _rePerpWeight := _reFrontal * _reRepulse * _creRightBias;

        yreDynGx := yreDynGx + _rePerpX * _rePerpWeight;
        yreDynGy := yreDynGy + _rePerpY * _rePerpWeight;

    END_IF

END_FOR

yreAusgangsTest := _reRepulse;

IF yboStop THEN yreSpeedFactor := 0.0; END_IF

END_FUNCTION_BLOCK

// ---- POUs/HAWinoCore/05_Bahnplanung/FB_StatesTest.TcPOU
FUNCTION_BLOCK FB_StatesTest
VAR_INPUT
	xboVectorTargetReached : BOOL;  //kommt von Algo
	xinSatus : INT; //Gewerk 3 Regelung
END_VAR
VAR_OUTPUT
	yinControl : RobotControl; //SChnittstellte Gewerk 3
	ysTargetPosition : sPosition; //Schnittstelle Gewerk 3
	yinTargetMap : INT; //Vektorregelung Ziel
END_VAR
VAR
	sStates : sStatesForTest;
	tonDelayWait : TON;
	tonDelayTargetReach : TON;
	tonDelayGripper : TON;
END_VAR
VAR CONSTANT
	//Robby 3
	creTarget1X : REAL := 635.1;
	creTarget1Y : REAL := 2668.6;
	creTarget1Phi : REAL := 0.4;
	creTarget2X : REAL := 1060.3;
	creTarget2Y : REAL := 2672.3;
	creTarget2Phi : REAL := -179.6;
	
END_VAR

CASE sStates OF
	
	sStatesForTest.Target1Vektor : 
	Gripper.closeGripperCommand := FALSE;
		yinTargetMap := 1;
		IF xboVectorTargetReached THEN 
			sStates := sStatesForTest.Wait1;//CoordinatesInFrontOfTarget1;
		END_IF;
		
	sStatesForTest.CoordinatesInFrontOfTarget1 :
		ysTargetPosition.reX := creTarget1X - 100;
		ysTargetPosition.reY := creTarget1Y;
		ysTargetPosition.reWinkel := creTarget1Phi;
		IF xinSatus = 3 THEN 
			sStates := sStatesForTest.Wait1;
		END_IF;
		
	sStatesForTest.Wait1 : 
	
			ysTargetPosition.reY := creTarget1Y;
		ysTargetPosition.reWinkel := creTarget1Phi;
		ysTargetPosition.reX := creTarget1X;
		IF 	xinSatus = 1 AND tonDelayWait.Q THEN 
			sStates := sStatesForTest.Target1;
		END_IF
		
	sStatesForTest.Target1 :
		
		IF xinSatus = 3 THEN 
			sStates := sStatesForTest.Wait2;
		END_IF;
		
	sStatesForTest.Wait2 : 
		Gripper.closeGripperCommand := TRUE;
		ysTargetPosition.reX := creTarget1X - 100;
		IF 	xinSatus = 1 AND tonDelayWait.Q THEN 
			sStates := sStatesForTest.AfterTarget1;
		END_IF
		
	sStatesForTest.AfterTarget1 :
		
		IF xinSatus = 3 THEN 
			sStates := sStatesForTest.Target2Vector;
		END_IF;
		
	sStatesForTest.Target2Vector :
	
		yinTargetMap := 2;
		IF xboVectorTargetReached THEN 
			sStates := sStatesForTest.Wait3;//CoordinatesInFrontOfTarget2;
		END_IF;
		
	sStatesForTest.CoordinatesInFrontOfTarget2 :
		ysTargetPosition.reX := creTarget2X + 100;
		ysTargetPosition.reY := creTarget2Y;
		ysTargetPosition.reWinkel := creTarget2Phi;
		IF xinSatus = 3 THEN 
			sStates := sStatesForTest.Wait3;
		END_IF;
		
		sStatesForTest.Wait3 : 
		ysTargetPosition.reY := creTarget2Y;
		ysTargetPosition.reWinkel := creTarget2Phi;
		ysTargetPosition.reX := creTarget2X;
		IF 	xinSatus = 1 AND tonDelayWait.Q THEN 
			sStates := sStatesForTest.Target2;
		END_IF	
		
	sStatesForTest.Target2 :
	
		
		IF xinSatus = 3 THEN 
			sStates := sStatesForTest.Wait4;
		END_IF;
		
		
		sStatesForTest.Wait4 : 
		Gripper.closeGripperCommand := FALSE;
		ysTargetPosition.reX := creTarget2X + 100;
		IF 	xinSatus = 1 AND tonDelayWait.Q THEN 
			sStates := sStatesForTest.AfterTarget2;
		END_IF	

	sStatesForTest.AfterTarget2 :
	
		IF xinSatus = 3 THEN 
			sStates := sStatesForTest.ParkingVector;
		END_IF;
		
	sStatesForTest.ParkingVector :
	
		yinTargetMap := 7;
		IF xboVectorTargetReached THEN 
			sStates := sStatesForTest.Finished;
		END_IF;
		
	sStatesForTest.Finished : ;
	
END_CASE

tonDelayWait(IN := (sStatesForTest.Wait1 = sStates) OR (sStatesForTest.Wait2 = sStates) OR (sStatesForTest.Wait3 = sStates) OR (sStatesForTest.Wait4 = sStates), PT := T#0.4S);

IF (sStatesForTest.Target1Vektor = sStates) OR (sStatesForTest.Target2Vector = sStates) OR (sStatesForTest.ParkingVector = sStates) THEN
	yinControl := 3;
END_IF

IF (sStatesForTest.CoordinatesInFrontOfTarget1 = sStates) OR (sStatesForTest.Target1 = sStates) OR (sStatesForTest.AfterTarget1 = sStates)
 OR (sStatesForTest.CoordinatesInFrontOfTarget2 = sStates) OR (sStatesForTest.Target2 = sStates) OR (sStatesForTest.AfterTarget2 = sStates) THEN
	yinControl := 4;
END_IF

IF (sStatesForTest.Finished = sStates) THEN
	yinControl := 1;
END_IF

IF (sStatesForTest.Wait1 = sStates) OR (sStatesForTest.Wait2 = sStates) OR (sStatesForTest.Wait3 = sStates) OR (sStatesForTest.Wait4 = sStates) THEN
	yinControl := 0;
END_IF

END_FUNCTION_BLOCK
